KUKA KRL program: EPS_2_251315_MH05A_A_20251118013654.src

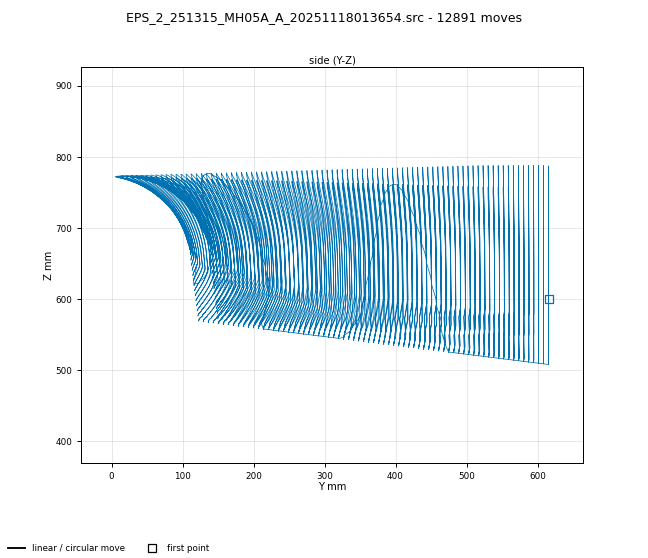
[picture p0: tool path of EPS_2_251315_MH05A_A_20251118013654.src, 12891 of 12893 moves have a stored position in this frame; points joined in program order, loops and branches not executed]
&ACCESS RVP
&REL 4
&COMMENT QRS 19112012
&PARAM EDITMASK = *
DEF PART()
EXT BAS (BAS_COMMAND :IN,REAL :IN )
INT I
BAS (#INITMOV,0 )

;KUKA QRS Post kuka4.cps  Date:22-06-2017 !

File_ID=2909

QRS_PRE_INIT()

;Init var - Until changes are made in qrs_pre_init
Outlet_Square_prg=0
Inlet_1_Square_prg=0
Inlet_2_Square_prg=0
Inlet_3_Square_prg=0
Inlet_4_Square_prg=0
Inlet_5_Square_prg=0

Outlet_1={X 0.000, Y 519.160, Z 687.500, B 0.000, E1 0.000 }
Inlet_1={X 0.000, Y 521.300, Z 657.500, B 0.000, E1 184.000 }
Outlet_1_type=201
Inlet_1_type=201
;QRS#1=Sidecore dimensions
;QRS#2=200-8" PVC SDR 35
;QRS#3=200-8" PVC SDR 35
;QRS#4=
;QRS#5=
;QRS#6=
;QRS#7=
;QRS#8=
;QRS#9=12-08 PSX
;QRS#10=12-08 PSX
;QRS#11=
;QRS#12=
;QRS#13=
;QRS#14=
;QRS#15=
;QRS#16=1220x127x1067 3,5'
;QRS#17=EPS Height
;QRS#18=788
;QRS#19=*
;QRS#20= UPDATED VERSION 22-06-2017
;QRS#21=*
Outlet_Square=0100
Inlet_1_Square=0100
Inlet_2_Square=0
Inlet_3_Square=0
Inlet_4_Square=0
Inlet_5_Square=0
Mill_Square=1
Outlet_Square_Prg=204
Inlet_1_Square_prg=204

QRS_INIT()

$ADVANCE=5

; T1
PTP {E1 173.595,E2 173.595}
PTP {X 0,Y 615.505,A -85,B 0,C 180,E1 173.595,E2 173.595,E3 0,E4 0,E5 0,E6 0}
QRS_SPEED_INIT()
LIN {X 0,Y 615.505,Z 600,A -85,B 0,C 180,E1 173.595,E2 173.595,E3 0,E4 0,E5 0,E6 0} C_VEL
LIN {X 0,Y 615.505,Z 517.862,A -85,B 0,C 180,E1 173.595,E2 173.595} C_VEL
LIN {X 0,Y 615.505,Z 509.682,A -85,B 0,C 180,E1 173.595,E2 173.595} C_VEL
LIN {X 0,Y 615.489,Z 507.682,A -85,B 0,C 180,E1 173.409,E2 173.409} C_VEL
LIN {X 0,Y 615.481,Z 507.696,A -85,B 0,C 180,E1 170.801,E2 170.801} C_VEL
LIN {X 0,Y 615.479,Z 507.691,A -85,B 0,C 180,E1 168.139,E2 168.139} C_VEL
LIN {X 0,Y 615.488,Z 507.682,A -85,B 0,C 180,E1 165.451,E2 165.451} C_VEL
LIN {X 0,Y 615.478,Z 507.699,A -85,B 0,C 180,E1 162.729,E2 162.729} C_VEL
LIN {X 0,Y 615.477,Z 507.687,A -85,B 0,C 180,E1 159.967,E2 159.967} C_VEL
LIN {X 0,Y 615.481,Z 507.683,A -85,B 0,C 180,E1 157.652,E2 157.652} C_VEL
LIN {X 0,Y 615.479,Z 507.691,A -85,B 0,C 180,E1 155.008,E2 155.008} C_VEL
LIN {X 0,Y 615.482,Z 507.688,A -85,B 0,C 180,E1 152.084,E2 152.084} C_VEL
LIN {X 0,Y 615.476,Z 507.686,A -85,B 0,C 180,E1 149.839,E2 149.839} C_VEL
LIN {X 0,Y 615.484,Z 507.683,A -85,B 0,C 180,E1 147.542,E2 147.542} C_VEL
LIN {X 0,Y 615.49,Z 507.685,A -85,B 0,C 180,E1 145.185,E2 145.185} C_VEL
LIN {X 0,Y 615.483,Z 507.698,A -85,B 0,C 180,E1 142.757,E2 142.757} C_VEL
LIN {X 0,Y 615.478,Z 507.686,A -85,B 0,C 180,E1 139.91,E2 139.91} C_VEL
LIN {X 0,Y 615.478,Z 507.684,A -85,B 0,C 180,E1 137.646,E2 137.646} C_VEL
LIN {X 0,Y 615.481,Z 507.693,A -85,B 0,C 180,E1 134.93,E2 134.93} C_VEL
LIN {X 0,Y 615.488,Z 507.687,A -85,B 0,C 180,E1 132.08,E2 132.08} C_VEL
LIN {X 0,Y 615.477,Z 507.685,A -85,B 0,C 180,E1 129.75,E2 129.75} C_VEL
LIN {X 0,Y 615.489,Z 507.691,A -85,B 0,C 180,E1 126.936,E2 126.936} C_VEL
LIN {X 0,Y 615.487,Z 507.686,A -85,B 0,C 180,E1 124.021,E2 124.021} C_VEL
LIN {X 0,Y 615.477,Z 507.684,A -85,B 0,C 180,E1 121.685,E2 121.685} C_VEL
LIN {X 0,Y 615.478,Z 507.685,A -85,B 0,C 180,E1 119.406,E2 119.406} C_VEL
LIN {X 0,Y 615.492,Z 507.688,A -85,B 0,C 180,E1 117.045,E2 117.045} C_VEL
LIN {X 0,Y 615.495,Z 507.689,A -85,B 0,C 180,E1 114.271,E2 114.271} C_VEL
LIN {X 0,Y 615.48,Z 507.684,A -85,B 0,C 180,E1 111.432,E2 111.432} C_VEL
LIN {X 0,Y 615.494,Z 507.701,A -85,B 0,C 180,E1 108.605,E2 108.605} C_VEL
LIN {X 0,Y 615.486,Z 507.684,A -85,B 0,C 180,E1 105.905,E2 105.905} C_VEL
LIN {X 0,Y 615.492,Z 507.887,A -85,B 0,C 180,E1 105.183,E2 105.183} C_VEL
LIN {X 0,Y 615.493,Z 525.05,A -85,B 0,C 180,E1 102.362,E2 102.362} C_VEL
LIN {X 0,Y 615.477,Z 542.524,A -85,B 0,C 180,E1 99.53,E2 99.53} C_VEL
LIN {X 0,Y 615.491,Z 546.889,A -85,B 0,C 180,E1 98.826,E2 98.826} C_VEL
LIN {X 0,Y 615.477,Z 653.781,A -85,B 0,C 180,E1 97.545,E2 97.545} C_VEL
LIN {X 0,Y 615.484,Z 666.943,A -85,B 0,C 180,E1 97.257,E2 97.257} C_VEL
LIN {X 0,Y 615.485,Z 679.264,A -85,B 0,C 180,E1 96.855,E2 96.855} C_VEL
LIN {X 0,Y 615.49,Z 691.591,A -85,B 0,C 180,E1 96.31,E2 96.31} C_VEL
LIN {X 0,Y 615.487,Z 702.986,A -85,B 0,C 180,E1 95.652,E2 95.652} C_VEL
LIN {X 0,Y 615.498,Z 713.247,A -85,B 0,C 180,E1 94.913,E2 94.913} C_VEL
LIN {X 0,Y 615.499,Z 722.526,A -85,B 0,C 180,E1 94.092,E2 94.092} C_VEL
LIN {X 0,Y 615.497,Z 731.469,A -85,B 0,C 180,E1 93.109,E2 93.109} C_VEL
LIN {X 0,Y 615.497,Z 738.692,A -85,B 0,C 180,E1 92.127,E2 92.127} C_VEL
LIN {X 0,Y 615.495,Z 745.319,A -85,B 0,C 180,E1 90.981,E2 90.981} C_VEL
LIN {X 0,Y 615.496,Z 749.706,A -85,B 0,C 180,E1 90,E2 90} C_VEL
LIN {X 0,Y 615.496,Z 752.021,A -85,B 0,C 180,E1 89.346,E2 89.346} C_VEL
LIN {X 0,Y 615.495,Z 753.917,A -85,B 0,C 180,E1 88.691,E2 88.691} C_VEL
LIN {X 0,Y 615.5,Z 755.401,A -85,B 0,C 180,E1 88.037,E2 88.037} C_VEL
LIN {X 0,Y 615.495,Z 757.09,A -85,B 0,C 180,E1 86.727,E2 86.727} C_VEL
LIN {X 0,Y 615.496,Z 757.254,A -85,B 0,C 180,E1 85.416,E2 85.416} C_VEL
LIN {X 0,Y 615.497,Z 755.79,A -85,B 0,C 180,E1 84.102,E2 84.102} C_VEL
LIN {X 0,Y 615.495,Z 754.424,A -85,B 0,C 180,E1 83.419,E2 83.419} C_VEL
LIN {X 0,Y 615.496,Z 751.671,A -85,B 0,C 180,E1 82.455,E2 82.455} C_VEL
LIN {X 0,Y 615.496,Z 747.841,A -85,B 0,C 180,E1 81.464,E2 81.464} C_VEL
LIN {X 0,Y 615.496,Z 742.869,A -85,B 0,C 180,E1 80.47,E2 80.47} C_VEL
LIN {X 0,Y 615.496,Z 736.598,A -85,B 0,C 180,E1 79.473,E2 79.473} C_VEL
LIN {X 0,Y 615.496,Z 728.708,A -85,B 0,C 180,E1 78.474,E2 78.474} C_VEL
LIN {X 0,Y 615.498,Z 720.622,A -85,B 0,C 180,E1 77.638,E2 77.638} C_VEL
LIN {X 0,Y 615.499,Z 710.724,A -85,B 0,C 180,E1 76.799,E2 76.799} C_VEL
LIN {X 0,Y 615.491,Z 699.961,A -85,B 0,C 180,E1 76.068,E2 76.068} C_VEL
LIN {X 0,Y 615.49,Z 688.509,A -85,B 0,C 180,E1 75.451,E2 75.451} C_VEL
LIN {X 0,Y 615.499,Z 676.28,A -85,B 0,C 180,E1 74.944,E2 74.944} C_VEL
LIN {X 0,Y 615.479,Z 663.455,A -85,B 0,C 180,E1 74.562,E2 74.562} C_VEL
LIN {X 0,Y 615.478,Z 649.799,A -85,B 0,C 180,E1 74.307,E2 74.307} C_VEL
LIN {X 0,Y 615.49,Z 546.948,A -85,B 0,C 180,E1 73.094,E2 73.094} C_VEL
LIN {X 0,Y 615.476,Z 529.77,A -85,B 0,C 180,E1 70.315,E2 70.315} C_VEL
LIN {X 0,Y 615.49,Z 513.503,A -85,B 0,C 180,E1 67.654,E2 67.654} C_VEL
LIN {X 0,Y 615.483,Z 507.686,A -85,B 0,C 180,E1 66.667,E2 66.667} C_VEL
LIN {X 0,Y 615.477,Z 507.684,A -85,B 0,C 180,E1 64.284,E2 64.284} C_VEL
LIN {X 0,Y 615.488,Z 507.694,A -85,B 0,C 180,E1 61.55,E2 61.55} C_VEL
LIN {X 0,Y 615.489,Z 507.689,A -85,B 0,C 180,E1 58.915,E2 58.915} C_VEL
LIN {X 0,Y 615.479,Z 507.684,A -85,B 0,C 180,E1 56.468,E2 56.468} C_VEL
LIN {X 0,Y 615.495,Z 507.692,A -85,B 0,C 180,E1 53.577,E2 53.577} C_VEL
LIN {X 0,Y 615.488,Z 507.69,A -85,B 0,C 180,E1 50.938,E2 50.938} C_VEL
LIN {X 0,Y 615.483,Z 507.684,A -85,B 0,C 180,E1 48.527,E2 48.527} C_VEL
LIN {X 0,Y 615.492,Z 507.686,A -85,B 0,C 180,E1 45.852,E2 45.852} C_VEL
LIN {X 0,Y 615.486,Z 507.693,A -85,B 0,C 180,E1 43.049,E2 43.049} C_VEL
LIN {X 0,Y 615.483,Z 507.684,A -85,B 0,C 180,E1 40.607,E2 40.607} C_VEL
LIN {X 0,Y 615.478,Z 507.686,A -85,B 0,C 180,E1 38.013,E2 38.013} C_VEL
LIN {X 0,Y 615.498,Z 507.691,A -85,B 0,C 180,E1 35.615,E2 35.615} C_VEL
LIN {X 0,Y 615.491,Z 507.698,A -85,B 0,C 180,E1 33.236,E2 33.236} C_VEL
LIN {X 0,Y 615.485,Z 507.69,A -85,B 0,C 180,E1 30.92,E2 30.92} C_VEL
LIN {X 0,Y 615.483,Z 507.683,A -85,B 0,C 180,E1 28.452,E2 28.452} C_VEL
LIN {X 0,Y 615.493,Z 507.693,A -85,B 0,C 180,E1 25.573,E2 25.573} C_VEL
LIN {X 0,Y 615.482,Z 507.688,A -85,B 0,C 180,E1 22.845,E2 22.845} C_VEL
LIN {X 0,Y 615.486,Z 507.683,A -85,B 0,C 180,E1 20.56,E2 20.56} C_VEL
LIN {X 0,Y 615.478,Z 507.687,A -85,B 0,C 180,E1 17.957,E2 17.957} C_VEL
LIN {X 0,Y 615.483,Z 507.699,A -85,B 0,C 180,E1 15.226,E2 15.226} C_VEL
LIN {X 0,Y 615.49,Z 507.682,A -85,B 0,C 180,E1 12.53,E2 12.53} C_VEL
LIN {X 0,Y 615.479,Z 507.689,A -85,B 0,C 180,E1 9.862,E2 9.862} C_VEL
LIN {X 0,Y 615.486,Z 507.697,A -85,B 0,C 180,E1 7.216,E2 7.216} C_VEL
LIN {X 0,Y 615.495,Z 507.681,A -85,B 0,C 180,E1 4.585,E2 4.585} C_VEL
LIN {X 0,Y 615.477,Z 507.688,A -85,B 0,C 180,E1 1.963,E2 1.963} C_VEL
LIN {X 0,Y 615.485,Z 507.702,A -85,B 0,C 180,E1 -0.654,E2 -0.654} C_VEL
LIN {X 0,Y 615.484,Z 507.685,A -85,B 0,C 180,E1 -3.273,E2 -3.273} C_VEL
LIN {X 0,Y 615.478,Z 507.686,A -85,B 0,C 180,E1 -5.899,E2 -5.899} C_VEL
LIN {X 0,Y 615.492,Z 507.699,A -85,B 0,C 180,E1 -8.537,E2 -8.537} C_VEL
LIN {X 0,Y 615.478,Z 507.687,A -85,B 0,C 180,E1 -11.193,E2 -11.193} C_VEL
LIN {X 0,Y 615.474,Z 507.687,A -85,B 0,C 180,E1 -13.933,E2 -13.933} C_VEL
LIN {X 0,Y 615.489,Z 507.702,A -85,B 0,C 180,E1 -16.587,E2 -16.587} C_VEL
LIN {X 0,Y 615.48,Z 507.685,A -85,B 0,C 180,E1 -19.338,E2 -19.338} C_VEL
LIN {X 0,Y 615.477,Z 507.691,A -85,B 0,C 180,E1 -22.137,E2 -22.137} C_VEL
LIN {X 0,Y 615.479,Z 507.691,A -85,B 0,C 180,E1 -24.992,E2 -24.992} C_VEL
LIN {X 0,Y 615.482,Z 507.686,A -85,B 0,C 180,E1 -27.915,E2 -27.915} C_VEL
LIN {X 0,Y 615.476,Z 507.692,A -85,B 0,C 180,E1 -30.161,E2 -30.161} C_VEL
LIN {X 0,Y 615.487,Z 507.699,A -85,B 0,C 180,E1 -32.458,E2 -32.458} C_VEL
LIN {X 0,Y 615.49,Z 507.693,A -85,B 0,C 180,E1 -34.815,E2 -34.815} C_VEL
LIN {X 0,Y 615.475,Z 507.687,A -85,B 0,C 180,E1 -37.243,E2 -37.243} C_VEL
LIN {X 0,Y 615.482,Z 507.689,A -85,B 0,C 180,E1 -40.09,E2 -40.09} C_VEL
LIN {X 0,Y 615.478,Z 507.697,A -85,B 0,C 180,E1 -42.354,E2 -42.354} C_VEL
LIN {X 0,Y 615.48,Z 507.689,A -85,B 0,C 180,E1 -45.069,E2 -45.069} C_VEL
LIN {X 0,Y 615.488,Z 507.685,A -85,B 0,C 180,E1 -47.92,E2 -47.92} C_VEL
LIN {X 0,Y 615.48,Z 507.694,A -85,B 0,C 180,E1 -50.25,E2 -50.25} C_VEL
LIN {X 0,Y 615.482,Z 507.688,A -85,B 0,C 180,E1 -53.064,E2 -53.064} C_VEL
LIN {X 0,Y 615.487,Z 507.686,A -85,B 0,C 180,E1 -55.979,E2 -55.979} C_VEL
LIN {X 0,Y 615.489,Z 507.69,A -85,B 0,C 180,E1 -58.914,E2 -58.914} C_VEL
LIN {X 0,Y 615.481,Z 507.683,A -85,B 0,C 180,E1 -61.551,E2 -61.551} C_VEL
LIN {X 0,Y 615.477,Z 507.696,A -85,B 0,C 180,E1 -64.284,E2 -64.284} C_VEL
LIN {X 0,Y 615.486,Z 507.7,A -85,B 0,C 180,E1 -66.444,E2 -66.444} C_VEL
LIN {X 0,Y 615.491,Z 507.764,A -85,B 0,C 180,E1 -67.838,E2 -67.838} C_VEL
LIN {X 0,Y 615.483,Z 528.08,A -85,B 0,C 180,E1 -70.662,E2 -70.662} C_VEL
LIN {X 0,Y 615.477,Z 548.189,A -85,B 0,C 180,E1 -73.414,E2 -73.414} C_VEL
LIN {X 0,Y 615.487,Z 568.274,A -85,B 0,C 180,E1 -76.126,E2 -76.126} C_VEL
LIN {X 0,Y 615.486,Z 575.644,A -85,B 0,C 180,E1 -77.114,E2 -77.114} C_VEL
LIN {X 0,Y 615.477,Z 683.848,A -85,B 0,C 180,E1 -78.411,E2 -78.411} C_VEL
LIN {X 0,Y 615.482,Z 696.355,A -85,B 0,C 180,E1 -78.682,E2 -78.682} C_VEL
LIN {X 0,Y 615.497,Z 709.489,A -85,B 0,C 180,E1 -79.108,E2 -79.108} C_VEL
LIN {X 0,Y 615.48,Z 721.483,A -85,B 0,C 180,E1 -79.64,E2 -79.64} C_VEL
LIN {X 0,Y 615.481,Z 733,A -85,B 0,C 180,E1 -80.304,E2 -80.304} C_VEL
LIN {X 0,Y 615.499,Z 743.344,A -85,B 0,C 180,E1 -81.05,E2 -81.05} C_VEL
LIN {X 0,Y 615.497,Z 751.814,A -85,B 0,C 180,E1 -81.794,E2 -81.794} C_VEL
LIN {X 0,Y 615.498,Z 759.608,A -85,B 0,C 180,E1 -82.62,E2 -82.62} C_VEL
LIN {X 0,Y 615.496,Z 767.204,A -85,B 0,C 180,E1 -83.608,E2 -83.608} C_VEL
LIN {X 0,Y 615.498,Z 774.205,A -85,B 0,C 180,E1 -84.759,E2 -84.759} C_VEL
LIN {X 0,Y 615.493,Z 778.852,A -85,B 0,C 180,E1 -85.744,E2 -85.744} C_VEL
LIN {X 0,Y 615.495,Z 782.399,A -85,B 0,C 180,E1 -86.727,E2 -86.727} C_VEL
LIN {X 0,Y 615.497,Z 784.233,A -85,B 0,C 180,E1 -87.382,E2 -87.382} C_VEL
LIN {X 0,Y 615.496,Z 785.608,A -85,B 0,C 180,E1 -88.037,E2 -88.037} C_VEL
LIN {X 0,Y 615.496,Z 787.174,A -85,B 0,C 180,E1 -89.346,E2 -89.346} C_VEL
LIN {X 0,Y 615.494,Z 787.389,A -85,B 0,C 180,E1 -90,E2 -90} C_VEL
LIN {X 0,Y 615.496,Z 786.58,A -85,B 0,C 180,E1 -91.309,E2 -91.309} C_VEL
LIN {X 0,Y 615.496,Z 785.608,A -85,B 0,C 180,E1 -91.963,E2 -91.963} C_VEL
LIN {X 0,Y 615.497,Z 784.233,A -85,B 0,C 180,E1 -92.618,E2 -92.618} C_VEL
LIN {X 0,Y 615.496,Z 781.35,A -85,B 0,C 180,E1 -93.601,E2 -93.601} C_VEL
LIN {X 0,Y 615.498,Z 777.442,A -85,B 0,C 180,E1 -94.584,E2 -94.584} C_VEL
LIN {X 0,Y 615.499,Z 772.406,A -85,B 0,C 180,E1 -95.57,E2 -95.57} C_VEL
LIN {X 0,Y 615.497,Z 765.869,A -85,B 0,C 180,E1 -96.583,E2 -96.583} C_VEL
LIN {X 0,Y 615.497,Z 758.135,A -85,B 0,C 180,E1 -97.545,E2 -97.545} C_VEL
LIN {X 0,Y 615.498,Z 750.047,A -85,B 0,C 180,E1 -98.371,E2 -98.371} C_VEL
LIN {X 0,Y 615.499,Z 740.17,A -85,B 0,C 180,E1 -99.198,E2 -99.198} C_VEL
LIN {X 0,Y 615.483,Z 728.986,A -85,B 0,C 180,E1 -99.945,E2 -99.945} C_VEL
LIN {X 0,Y 615.481,Z 718.029,A -85,B 0,C 180,E1 -100.527,E2 -100.527} C_VEL
LIN {X 0,Y 615.499,Z 705.423,A -85,B 0,C 180,E1 -101.042,E2 -101.042} C_VEL
LIN {X 0,Y 615.479,Z 693.079,A -85,B 0,C 180,E1 -101.401,E2 -101.401} C_VEL
LIN {X 0,Y 615.477,Z 679.489,A -85,B 0,C 180,E1 -101.652,E2 -101.652} C_VEL
LIN {X 0,Y 615.486,Z 575.644,A -85,B 0,C 180,E1 -102.886,E2 -102.886} C_VEL
LIN {X 0,Y 615.479,Z 554.469,A -85,B 0,C 180,E1 -105.735,E2 -105.735} C_VEL
LIN {X 0,Y 615.479,Z 534.609,A -85,B 0,C 180,E1 -108.44,E2 -108.44} C_VEL
LIN {X 0,Y 615.497,Z 514.243,A -85,B 0,C 180,E1 -111.255,E2 -111.255} C_VEL
LIN {X 0,Y 615.489,Z 507.683,A -85,B 0,C 180,E1 -112.188,E2 -112.188} C_VEL
LIN {X 0,Y 615.488,Z 507.687,A -85,B 0,C 180,E1 -114.991,E2 -114.991} C_VEL
LIN {X 0,Y 615.483,Z 507.69,A -85,B 0,C 180,E1 -117.915,E2 -117.915} C_VEL
LIN {X 0,Y 615.499,Z 507.681,A -85,B 0,C 180,E1 -120.159,E2 -120.159} C_VEL
LIN {X 0,Y 615.481,Z 507.683,A -85,B 0,C 180,E1 -122.457,E2 -122.457} C_VEL
LIN {X 0,Y 615.478,Z 507.686,A -85,B 0,C 180,E1 -124.815,E2 -124.815} C_VEL
LIN {X 0,Y 615.496,Z 507.693,A -85,B 0,C 180,E1 -127.241,E2 -127.241} C_VEL
LIN {X 0,Y 615.49,Z 507.684,A -85,B 0,C 180,E1 -130.089,E2 -130.089} C_VEL
LIN {X 0,Y 615.49,Z 507.681,A -85,B 0,C 180,E1 -132.351,E2 -132.351} C_VEL
LIN {X 0,Y 615.481,Z 507.691,A -85,B 0,C 180,E1 -135.068,E2 -135.068} C_VEL
LIN {X 0,Y 615.477,Z 507.69,A -85,B 0,C 180,E1 -137.919,E2 -137.919} C_VEL
LIN {X 0,Y 615.498,Z 507.68,A -85,B 0,C 180,E1 -140.251,E2 -140.251} C_VEL
LIN {X 0,Y 615.48,Z 507.691,A -85,B 0,C 180,E1 -143.063,E2 -143.063} C_VEL
LIN {X 0,Y 615.494,Z 507.695,A -85,B 0,C 180,E1 -145.297,E2 -145.297} C_VEL
LIN {X 0,Y 615.485,Z 507.683,A -85,B 0,C 180,E1 -148.314,E2 -148.314} C_VEL
LIN {X 0,Y 615.482,Z 507.683,A -85,B 0,C 180,E1 -150.593,E2 -150.593} C_VEL
LIN {X 0,Y 615.478,Z 507.689,A -85,B 0,C 180,E1 -152.954,E2 -152.954} C_VEL
LIN {X 0,Y 615.478,Z 507.695,A -85,B 0,C 180,E1 -155.728,E2 -155.728} C_VEL
LIN {X 0,Y 615.486,Z 507.682,A -85,B 0,C 180,E1 -158.568,E2 -158.568} C_VEL
LIN {X 0,Y 615.495,Z 507.699,A -85,B 0,C 180,E1 -161.389,E2 -161.389} C_VEL
LIN {X 0,Y 615.48,Z 507.686,A -85,B 0,C 180,E1 -164.095,E2 -164.095} C_VEL
LIN {X 0,Y 615.478,Z 507.687,A -85,B 0,C 180,E1 -166.799,E2 -166.799} C_VEL
LIN {X 0,Y 615.488,Z 507.701,A -85,B 0,C 180,E1 -169.473,E2 -169.473} C_VEL
LIN {X 0,Y 615.479,Z 507.686,A -85,B 0,C 180,E1 -172.124,E2 -172.124} C_VEL
LIN {X 0,Y 615.481,Z 507.685,A -85,B 0,C 180,E1 -174.759,E2 -174.759} C_VEL
LIN {X 0,Y 615.495,Z 507.699,A -85,B 0,C 180,E1 -177.382,E2 -177.382} C_VEL
LIN {X 0,Y 615.477,Z 507.688,A -85,B 0,C 180,E1 -180,E2 -180} C_VEL
LIN {X 0,Y 615.492,Z 507.682,A -85,B 0,C 180,E1 -182.618,E2 -182.618} C_VEL
LIN {X 0,Y 615.481,Z 507.697,A -85,B 0,C 180,E1 -185.241,E2 -185.241} C_VEL
LIN {X 0,Y 615.489,Z 507.682,A -85,B 0,C 180,E1 -186.591,E2 -186.591} C_VEL
LIN {X 0,Y 614.809,Z 507.843,A -85,B 0,C 180,E1 -187.137,E2 -187.137} C_VEL
LIN {X 0,Y 611.97,Z 508.251,A -85,B 0,C 180,E1 -188.023,E2 -188.023} C_VEL
LIN {X 0,Y 609.577,Z 508.566,A -85,B 0,C 180,E1 -188.735,E2 -188.735} C_VEL
LIN {X 0,Y 608.542,Z 508.685,A -85,B 0,C 180,E1 -189.285,E2 -189.285} C_VEL
LIN {X 0,Y 608.452,Z 508.693,A -85,B 0,C 180,E1 -189.471,E2 -189.471} C_VEL
LIN {X 0,Y 608.456,Z 508.689,A -85,B 0,C 180,E1 -192,E2 -192} C_VEL
LIN {X 0,Y 608.474,Z 508.685,A -85,B 0,C 180,E1 -194.721,E2 -194.721} C_VEL
LIN {X 0,Y 608.445,Z 508.698,A -85,B 0,C 180,E1 -197.477,E2 -197.477} C_VEL
LIN {X 0,Y 608.458,Z 508.687,A -85,B 0,C 180,E1 -200.275,E2 -200.275} C_VEL
LIN {X 0,Y 608.449,Z 508.687,A -85,B 0,C 180,E1 -202.477,E2 -202.477} C_VEL
LIN {X 0,Y 608.453,Z 508.696,A -85,B 0,C 180,E1 -205.301,E2 -205.301} C_VEL
LIN {X 0,Y 608.446,Z 508.697,A -85,B 0,C 180,E1 -207.518,E2 -207.518} C_VEL
LIN {X 0,Y 608.465,Z 508.688,A -85,B 0,C 180,E1 -209.973,E2 -209.973} C_VEL
LIN {X 0,Y 608.458,Z 508.686,A -85,B 0,C 180,E1 -212.524,E2 -212.524} C_VEL
LIN {X 0,Y 608.453,Z 508.696,A -85,B 0,C 180,E1 -215.277,E2 -215.277} C_VEL
LIN {X 0,Y 608.464,Z 508.691,A -85,B 0,C 180,E1 -217.747,E2 -217.747} C_VEL
LIN {X 0,Y 608.446,Z 508.688,A -85,B 0,C 180,E1 -220.33,E2 -220.33} C_VEL
LIN {X 0,Y 608.467,Z 508.695,A -85,B 0,C 180,E1 -223.31,E2 -223.31} C_VEL
LIN {X 0,Y 608.469,Z 508.686,A -85,B 0,C 180,E1 -226.132,E2 -226.132} C_VEL
LIN {X 0,Y 608.452,Z 508.689,A -85,B 0,C 180,E1 -228.824,E2 -228.824} C_VEL
LIN {X 0,Y 608.468,Z 508.696,A -85,B 0,C 180,E1 -231.413,E2 -231.413} C_VEL
LIN {X 0,Y 608.458,Z 508.689,A -85,B 0,C 180,E1 -233.954,E2 -233.954} C_VEL
LIN {X 0,Y 608.449,Z 508.688,A -85,B 0,C 180,E1 -236.329,E2 -236.329} C_VEL
LIN {X 0,Y 608.461,Z 508.687,A -85,B 0,C 180,E1 -238.731,E2 -238.731} C_VEL
LIN {X 0,Y 608.475,Z 508.695,A -85,B 0,C 180,E1 -241.381,E2 -241.381} C_VEL
LIN {X 0,Y 608.443,Z 508.69,A -85,B 0,C 180,E1 -243.965,E2 -243.965} C_VEL
LIN {X 0,Y 608.467,Z 508.686,A -85,B 0,C 180,E1 -246.156,E2 -246.156} C_VEL
LIN {X 0,Y 608.469,Z 508.685,A -85,B 0,C 180,E1 -248.309,E2 -248.309} C_VEL
LIN {X 0,Y 608.477,Z 508.693,A -85,B 0,C 180,E1 -251.284,E2 -251.284} C_VEL
LIN {X 0,Y 608.463,Z 508.689,A -85,B 0,C 180,E1 -253.907,E2 -253.907} C_VEL
LIN {X 0,Y 608.483,Z 508.758,A -85,B 0,C 180,E1 -254.723,E2 -254.723} C_VEL
LIN {X 0,Y 608.493,Z 525.455,A -85,B 0,C 180,E1 -257.493,E2 -257.493} C_VEL
LIN {X 0,Y 608.473,Z 541.956,A -85,B 0,C 180,E1 -260.191,E2 -260.191} C_VEL
LIN {X 0,Y 608.475,Z 547.189,A -85,B 0,C 180,E1 -261.04,E2 -261.04} C_VEL
LIN {X 0,Y 608.523,Z 654.213,A -85,B 0,C 180,E1 -262.326,E2 -262.326} C_VEL
LIN {X 0,Y 608.519,Z 667.268,A -85,B 0,C 180,E1 -262.618,E2 -262.618} C_VEL
LIN {X 0,Y 608.509,Z 680.713,A -85,B 0,C 180,E1 -263.068,E2 -263.068} C_VEL
LIN {X 0,Y 608.502,Z 692.957,A -85,B 0,C 180,E1 -263.635,E2 -263.635} C_VEL
LIN {X 0,Y 608.485,Z 703.909,A -85,B 0,C 180,E1 -264.283,E2 -264.283} C_VEL
LIN {X 0,Y 608.476,Z 714.098,A -85,B 0,C 180,E1 -265.031,E2 -265.031} C_VEL
LIN {X 0,Y 608.473,Z 723.296,A -85,B 0,C 180,E1 -265.86,E2 -265.86} C_VEL
LIN {X 0,Y 608.459,Z 732.223,A -85,B 0,C 180,E1 -266.855,E2 -266.855} C_VEL
LIN {X 0,Y 608.454,Z 739.435,A -85,B 0,C 180,E1 -267.849,E2 -267.849} C_VEL
LIN {X 0,Y 608.449,Z 744.316,A -85,B 0,C 180,E1 -268.676,E2 -268.676} C_VEL
LIN {X 0,Y 608.442,Z 749.071,A -85,B 0,C 180,E1 -269.669,E2 -269.669} C_VEL
LIN {X 0,Y 608.439,Z 752.725,A -85,B 0,C 180,E1 -270.662,E2 -270.662} C_VEL
LIN {X 0,Y 608.447,Z 754.616,A -85,B 0,C 180,E1 -271.324,E2 -271.324} C_VEL
LIN {X 0,Y 608.445,Z 756.078,A -85,B 0,C 180,E1 -271.986,E2 -271.986} C_VEL
LIN {X 0,Y 608.421,Z 757.733,A -85,B 0,C 180,E1 -273.311,E2 -273.311} C_VEL
LIN {X 0,Y 608.433,Z 757.989,A -85,B 0,C 180,E1 -273.974,E2 -273.974} C_VEL
LIN {X 0,Y 608.429,Z 757.832,A -85,B 0,C 180,E1 -274.638,E2 -274.638} C_VEL
LIN {X 0,Y 608.434,Z 756.307,A -85,B 0,C 180,E1 -275.967,E2 -275.967} C_VEL
LIN {X 0,Y 608.448,Z 754.954,A -85,B 0,C 180,E1 -276.633,E2 -276.633} C_VEL
LIN {X 0,Y 608.427,Z 752.071,A -85,B 0,C 180,E1 -277.633,E2 -277.633} C_VEL
LIN {X 0,Y 608.43,Z 748.15,A -85,B 0,C 180,E1 -278.636,E2 -278.636} C_VEL
LIN {X 0,Y 608.435,Z 743.074,A -85,B 0,C 180,E1 -279.642,E2 -279.642} C_VEL
LIN {X 0,Y 608.443,Z 736.674,A -85,B 0,C 180,E1 -280.65,E2 -280.65} C_VEL
LIN {X 0,Y 608.474,Z 728.627,A -85,B 0,C 180,E1 -281.661,E2 -281.661} C_VEL
LIN {X 0,Y 608.468,Z 720.403,A -85,B 0,C 180,E1 -282.507,E2 -282.507} C_VEL
LIN {X 0,Y 608.481,Z 710.336,A -85,B 0,C 180,E1 -283.356,E2 -283.356} C_VEL
LIN {X 0,Y 608.489,Z 698.896,A -85,B 0,C 180,E1 -284.122,E2 -284.122} C_VEL
LIN {X 0,Y 608.518,Z 687.649,A -85,B 0,C 180,E1 -284.719,E2 -284.719} C_VEL
LIN {X 0,Y 608.545,Z 675.035,A -85,B 0,C 180,E1 -285.232,E2 -285.232} C_VEL
LIN {X 0,Y 608.545,Z 662.387,A -85,B 0,C 180,E1 -285.597,E2 -285.597} C_VEL
LIN {X 0,Y 608.547,Z 649.513,A -85,B 0,C 180,E1 -285.833,E2 -285.833} C_VEL
LIN {X 0,Y 608.467,Z 547.168,A -85,B 0,C 180,E1 -287.053,E2 -287.053} C_VEL
LIN {X 0,Y 608.488,Z 529.572,A -85,B 0,C 180,E1 -289.92,E2 -289.92} C_VEL
LIN {X 0,Y 608.512,Z 512.592,A -85,B 0,C 180,E1 -292.726,E2 -292.726} C_VEL
LIN {X 0,Y 608.464,Z 508.688,A -85,B 0,C 180,E1 -293.393,E2 -293.393} C_VEL
LIN {X 0,Y 608.443,Z 508.69,A -85,B 0,C 180,E1 -296.035,E2 -296.035} C_VEL
LIN {X 0,Y 608.475,Z 508.694,A -85,B 0,C 180,E1 -298.619,E2 -298.619} C_VEL
LIN {X 0,Y 608.46,Z 508.688,A -85,B 0,C 180,E1 -301.316,E2 -301.316} C_VEL
LIN {X 0,Y 608.471,Z 508.685,A -85,B 0,C 180,E1 -303.734,E2 -303.734} C_VEL
LIN {X 0,Y 608.476,Z 508.686,A -85,B 0,C 180,E1 -306.089,E2 -306.089} C_VEL
LIN {X 0,Y 608.468,Z 508.694,A -85,B 0,C 180,E1 -308.587,E2 -308.587} C_VEL
LIN {X 0,Y 608.458,Z 508.688,A -85,B 0,C 180,E1 -311.341,E2 -311.341} C_VEL
LIN {X 0,Y 608.459,Z 508.69,A -85,B 0,C 180,E1 -314.264,E2 -314.264} C_VEL
LIN {X 0,Y 608.452,Z 508.692,A -85,B 0,C 180,E1 -317.04,E2 -317.04} C_VEL
LIN {X 0,Y 608.446,Z 508.688,A -85,B 0,C 180,E1 -319.696,E2 -319.696} C_VEL
LIN {X 0,Y 608.463,Z 508.69,A -85,B 0,C 180,E1 -322.253,E2 -322.253} C_VEL
LIN {X 0,Y 608.481,Z 508.687,A -85,B 0,C 180,E1 -325.088,E2 -325.088} C_VEL
LIN {X 0,Y 608.463,Z 508.686,A -85,B 0,C 180,E1 -327.905,E2 -327.905} C_VEL
LIN {X 0,Y 608.472,Z 508.688,A -85,B 0,C 180,E1 -330.22,E2 -330.22} C_VEL
LIN {X 0,Y 608.474,Z 508.693,A -85,B 0,C 180,E1 -332.791,E2 -332.791} C_VEL
LIN {X 0,Y 608.445,Z 508.688,A -85,B 0,C 180,E1 -335.428,E2 -335.428} C_VEL
LIN {X 0,Y 608.471,Z 508.69,A -85,B 0,C 180,E1 -338.308,E2 -338.308} C_VEL
LIN {X 0,Y 608.469,Z 508.686,A -85,B 0,C 180,E1 -341.28,E2 -341.28} C_VEL
LIN {X 0,Y 608.456,Z 508.687,A -85,B 0,C 180,E1 -343.906,E2 -343.906} C_VEL
LIN {X 0,Y 608.457,Z 508.698,A -85,B 0,C 180,E1 -346.643,E2 -346.643} C_VEL
LIN {X 0,Y 608.463,Z 508.687,A -85,B 0,C 180,E1 -349.35,E2 -349.35} C_VEL
LIN {X 0,Y 608.471,Z 508.687,A -85,B 0,C 180,E1 -352.033,E2 -352.033} C_VEL
LIN {X 0,Y 608.461,Z 508.696,A -85,B 0,C 180,E1 -354.698,E2 -354.698} C_VEL
LIN {X 0,Y 608.481,Z 508.684,A -85,B 0,C 180,E1 -357.352,E2 -357.352} C_VEL
LIN {X 0,Y 608.467,Z 508.687,A -85,B 0,C 180,E1 -360,E2 -360} C_VEL
LIN {X 0,Y 608.484,Z 508.694,A -85,B 0,C 180,E1 -362.648,E2 -362.648} C_VEL
LIN {X 0,Y 608.46,Z 508.687,A -85,B 0,C 180,E1 -365.302,E2 -365.302} C_VEL
LIN {X 0,Y 608.472,Z 508.686,A -85,B 0,C 180,E1 -367.967,E2 -367.967} C_VEL
LIN {X 0,Y 608.463,Z 508.696,A -85,B 0,C 180,E1 -370.65,E2 -370.65} C_VEL
LIN {X 0,Y 608.455,Z 508.687,A -85,B 0,C 180,E1 -373.357,E2 -373.357} C_VEL
LIN {X 0,Y 608.455,Z 508.69,A -85,B 0,C 180,E1 -376.094,E2 -376.094} C_VEL
LIN {X 0,Y 608.452,Z 508.693,A -85,B 0,C 180,E1 -378.87,E2 -378.87} C_VEL
LIN {X 0,Y 608.464,Z 508.686,A -85,B 0,C 180,E1 -381.692,E2 -381.692} C_VEL
LIN {X 0,Y 608.445,Z 508.699,A -85,B 0,C 180,E1 -384.571,E2 -384.571} C_VEL
LIN {X 0,Y 608.47,Z 508.686,A -85,B 0,C 180,E1 -387.208,E2 -387.208} C_VEL
LIN {X 0,Y 608.464,Z 508.687,A -85,B 0,C 180,E1 -389.973,E2 -389.973} C_VEL
LIN {X 0,Y 608.46,Z 508.697,A -85,B 0,C 180,E1 -392.524,E2 -392.524} C_VEL
LIN {X 0,Y 608.449,Z 508.688,A -85,B 0,C 180,E1 -395.277,E2 -395.277} C_VEL
LIN {X 0,Y 608.462,Z 508.686,A -85,B 0,C 180,E1 -397.747,E2 -397.747} C_VEL
LIN {X 0,Y 608.45,Z 508.694,A -85,B 0,C 180,E1 -400.33,E2 -400.33} C_VEL
LIN {X 0,Y 608.463,Z 508.686,A -85,B 0,C 180,E1 -403.31,E2 -403.31} C_VEL
LIN {X 0,Y 608.471,Z 508.689,A -85,B 0,C 180,E1 -406.132,E2 -406.132} C_VEL
LIN {X 0,Y 608.458,Z 508.692,A -85,B 0,C 180,E1 -408.825,E2 -408.825} C_VEL
LIN {X 0,Y 608.465,Z 508.686,A -85,B 0,C 180,E1 -411.413,E2 -411.413} C_VEL
LIN {X 0,Y 608.457,Z 508.688,A -85,B 0,C 180,E1 -413.953,E2 -413.953} C_VEL
LIN {X 0,Y 608.467,Z 508.693,A -85,B 0,C 180,E1 -416.33,E2 -416.33} C_VEL
LIN {X 0,Y 608.477,Z 508.691,A -85,B 0,C 180,E1 -418.728,E2 -418.728} C_VEL
LIN {X 0,Y 608.467,Z 508.686,A -85,B 0,C 180,E1 -421.382,E2 -421.382} C_VEL
LIN {X 0,Y 608.438,Z 508.691,A -85,B 0,C 180,E1 -423.965,E2 -423.965} C_VEL
LIN {X 0,Y 608.469,Z 508.69,A -85,B 0,C 180,E1 -426.156,E2 -426.156} C_VEL
LIN {X 0,Y 608.472,Z 508.737,A -85,B 0,C 180,E1 -427.707,E2 -427.707} C_VEL
LIN {X 0,Y 608.535,Z 524.321,A -85,B 0,C 180,E1 -429.905,E2 -429.905} C_VEL
LIN {X 0,Y 608.527,Z 544.47,A -85,B 0,C 180,E1 -432.699,E2 -432.699} C_VEL
LIN {X 0,Y 608.497,Z 565.878,A -85,B 0,C 180,E1 -435.622,E2 -435.622} C_VEL
LIN {X 0,Y 608.495,Z 576.169,A -85,B 0,C 180,E1 -436.984,E2 -436.984} C_VEL
LIN {X 0,Y 608.534,Z 683.962,A -85,B 0,C 180,E1 -438.277,E2 -438.277} C_VEL
LIN {X 0,Y 608.533,Z 697.226,A -85,B 0,C 180,E1 -438.572,E2 -438.572} C_VEL
LIN {X 0,Y 608.544,Z 710.334,A -85,B 0,C 180,E1 -439.009,E2 -439.009} C_VEL
LIN {X 0,Y 608.498,Z 721.64,A -85,B 0,C 180,E1 -439.519,E2 -439.519} C_VEL
LIN {X 0,Y 608.471,Z 733.201,A -85,B 0,C 180,E1 -440.191,E2 -440.191} C_VEL
LIN {X 0,Y 608.485,Z 743.596,A -85,B 0,C 180,E1 -440.946,E2 -440.946} C_VEL
LIN {X 0,Y 608.475,Z 752.114,A -85,B 0,C 180,E1 -441.699,E2 -441.699} C_VEL
LIN {X 0,Y 608.471,Z 759.962,A -85,B 0,C 180,E1 -442.534,E2 -442.534} C_VEL
LIN {X 0,Y 608.46,Z 767.287,A -85,B 0,C 180,E1 -443.485,E2 -443.485} C_VEL
LIN {X 0,Y 608.45,Z 772.867,A -85,B 0,C 180,E1 -444.366,E2 -444.366} C_VEL
LIN {X 0,Y 608.432,Z 777.951,A -85,B 0,C 180,E1 -445.362,E2 -445.362} C_VEL
LIN {X 0,Y 608.449,Z 781.896,A -85,B 0,C 180,E1 -446.358,E2 -446.358} C_VEL
LIN {X 0,Y 608.425,Z 784.809,A -85,B 0,C 180,E1 -447.352,E2 -447.352} C_VEL
LIN {X 0,Y 608.441,Z 786.201,A -85,B 0,C 180,E1 -448.014,E2 -448.014} C_VEL
LIN {X 0,Y 608.438,Z 787.783,A -85,B 0,C 180,E1 -449.338,E2 -449.338} C_VEL
LIN {X 0,Y 608.434,Z 788,A -85,B 0,C 180,E1 -450,E2 -450} C_VEL
LIN {X 0,Y 608.448,Z 787.184,A -85,B 0,C 180,E1 -451.324,E2 -451.324} C_VEL
LIN {X 0,Y 608.441,Z 786.201,A -85,B 0,C 180,E1 -451.986,E2 -451.986} C_VEL
LIN {X 0,Y 608.425,Z 784.809,A -85,B 0,C 180,E1 -452.648,E2 -452.648} C_VEL
LIN {X 0,Y 608.449,Z 781.896,A -85,B 0,C 180,E1 -453.642,E2 -453.642} C_VEL
LIN {X 0,Y 608.432,Z 777.951,A -85,B 0,C 180,E1 -454.638,E2 -454.638} C_VEL
LIN {X 0,Y 608.437,Z 771.877,A -85,B 0,C 180,E1 -455.801,E2 -455.801} C_VEL
LIN {X 0,Y 608.462,Z 765.236,A -85,B 0,C 180,E1 -456.799,E2 -456.799} C_VEL
LIN {X 0,Y 608.455,Z 756.991,A -85,B 0,C 180,E1 -457.8,E2 -457.8} C_VEL
LIN {X 0,Y 608.472,Z 748.539,A -85,B 0,C 180,E1 -458.636,E2 -458.636} C_VEL
LIN {X 0,Y 608.474,Z 738.094,A -85,B 0,C 180,E1 -459.473,E2 -459.473} C_VEL
LIN {X 0,Y 608.482,Z 727.76,A -85,B 0,C 180,E1 -460.145,E2 -460.145} C_VEL
LIN {X 0,Y 608.521,Z 716.245,A -85,B 0,C 180,E1 -460.741,E2 -460.741} C_VEL
LIN {X 0,Y 608.528,Z 704.882,A -85,B 0,C 180,E1 -461.192,E2 -461.192} C_VEL
LIN {X 0,Y 608.535,Z 692.279,A -85,B 0,C 180,E1 -461.554,E2 -461.554} C_VEL
LIN {X 0,Y 608.535,Z 679.622,A -85,B 0,C 180,E1 -461.787,E2 -461.787} C_VEL
LIN {X 0,Y 608.495,Z 576.169,A -85,B 0,C 180,E1 -463.016,E2 -463.016} C_VEL
LIN {X 0,Y 608.487,Z 557.063,A -85,B 0,C 180,E1 -465.577,E2 -465.577} C_VEL
LIN {X 0,Y 608.516,Z 536.995,A -85,B 0,C 180,E1 -468.332,E2 -468.332} C_VEL
LIN {X 0,Y 608.572,Z 516.765,A -85,B 0,C 180,E1 -471.154,E2 -471.154} C_VEL
LIN {X 0,Y 608.455,Z 508.689,A -85,B 0,C 180,E1 -472.316,E2 -472.316} C_VEL
LIN {X 0,Y 608.455,Z 508.687,A -85,B 0,C 180,E1 -474.57,E2 -474.57} C_VEL
LIN {X 0,Y 608.484,Z 508.689,A -85,B 0,C 180,E1 -477.208,E2 -477.208} C_VEL
LIN {X 0,Y 608.467,Z 508.688,A -85,B 0,C 180,E1 -479.971,E2 -479.971} C_VEL
LIN {X 0,Y 608.457,Z 508.686,A -85,B 0,C 180,E1 -482.521,E2 -482.521} C_VEL
LIN {X 0,Y 608.443,Z 508.69,A -85,B 0,C 180,E1 -484.904,E2 -484.904} C_VEL
LIN {X 0,Y 608.471,Z 508.691,A -85,B 0,C 180,E1 -487.745,E2 -487.745} C_VEL
LIN {X 0,Y 608.45,Z 508.688,A -85,B 0,C 180,E1 -490.329,E2 -490.329} C_VEL
LIN {X 0,Y 608.485,Z 508.691,A -85,B 0,C 180,E1 -493.31,E2 -493.31} C_VEL
LIN {X 0,Y 608.466,Z 508.687,A -85,B 0,C 180,E1 -496.13,E2 -496.13} C_VEL
LIN {X 0,Y 608.449,Z 508.689,A -85,B 0,C 180,E1 -498.823,E2 -498.823} C_VEL
LIN {X 0,Y 608.465,Z 508.696,A -85,B 0,C 180,E1 -501.412,E2 -501.412} C_VEL
LIN {X 0,Y 608.472,Z 508.688,A -85,B 0,C 180,E1 -503.949,E2 -503.949} C_VEL
LIN {X 0,Y 608.462,Z 508.686,A -85,B 0,C 180,E1 -506.329,E2 -506.329} C_VEL
LIN {X 0,Y 608.469,Z 508.686,A -85,B 0,C 180,E1 -508.727,E2 -508.727} C_VEL
LIN {X 0,Y 608.471,Z 508.695,A -85,B 0,C 180,E1 -511.378,E2 -511.378} C_VEL
LIN {X 0,Y 608.475,Z 508.685,A -85,B 0,C 180,E1 -514.276,E2 -514.276} C_VEL
LIN {X 0,Y 608.447,Z 508.69,A -85,B 0,C 180,E1 -516.876,E2 -516.876} C_VEL
LIN {X 0,Y 608.464,Z 508.694,A -85,B 0,C 180,E1 -519.319,E2 -519.319} C_VEL
LIN {X 0,Y 608.448,Z 508.692,A -85,B 0,C 180,E1 -521.828,E2 -521.828} C_VEL
LIN {X 0,Y 608.463,Z 508.686,A -85,B 0,C 180,E1 -524.594,E2 -524.594} C_VEL
LIN {X 0,Y 608.473,Z 508.693,A -85,B 0,C 180,E1 -527.323,E2 -527.323} C_VEL
LIN {X 0,Y 608.45,Z 508.689,A -85,B 0,C 180,E1 -530.023,E2 -530.023} C_VEL
LIN {X 0,Y 608.474,Z 508.685,A -85,B 0,C 180,E1 -532.701,E2 -532.701} C_VEL
LIN {X 0,Y 608.464,Z 508.695,A -85,B 0,C 180,E1 -535.362,E2 -535.362} C_VEL
LIN {X 0,Y 608.446,Z 508.69,A -85,B 0,C 180,E1 -538.014,E2 -538.014} C_VEL
LIN {X 0,Y 608.478,Z 508.684,A -85,B 0,C 180,E1 -540.662,E2 -540.662} C_VEL
LIN {X 0,Y 608.478,Z 508.693,A -85,B 0,C 180,E1 -543.311,E2 -543.311} C_VEL
LIN {X 0,Y 608.453,Z 508.689,A -85,B 0,C 180,E1 -545.967,E2 -545.967} C_VEL
LIN {X 0,Y 608.457,Z 508.687,A -85,B 0,C 180,E1 -548.636,E2 -548.636} C_VEL
LIN {X 0,Y 608.452,Z 508.693,A -85,B 0,C 180,E1 -549.471,E2 -549.471} C_VEL
LIN {X 0,Y 607.772,Z 508.774,A -85,B 0,C 180,E1 -550.024,E2 -550.024} C_VEL
LIN {X 0,Y 604.917,Z 509.13,A -85,B 0,C 180,E1 -550.921,E2 -550.921} C_VEL
LIN {X 0,Y 602.516,Z 509.434,A -85,B 0,C 180,E1 -551.642,E2 -551.642} C_VEL
LIN {X 0,Y 601.488,Z 509.556,A -85,B 0,C 180,E1 -552.199,E2 -552.199} C_VEL
LIN {X 0,Y 601.406,Z 509.565,A -85,B 0,C 180,E1 -552.388,E2 -552.388} C_VEL
LIN {X 0,Y 601.426,Z 509.565,A -85,B 0,C 180,E1 -554.897,E2 -554.897} C_VEL
LIN {X 0,Y 601.426,Z 509.566,A -85,B 0,C 180,E1 -556.986,E2 -556.986} C_VEL
LIN {X 0,Y 601.402,Z 509.57,A -85,B 0,C 180,E1 -559.81,E2 -559.81} C_VEL
LIN {X 0,Y 601.406,Z 509.565,A -85,B 0,C 180,E1 -562.606,E2 -562.606} C_VEL
LIN {X 0,Y 601.399,Z 509.568,A -85,B 0,C 180,E1 -564.879,E2 -564.879} C_VEL
LIN {X 0,Y 601.417,Z 509.567,A -85,B 0,C 180,E1 -567.868,E2 -567.868} C_VEL
LIN {X 0,Y 601.441,Z 509.561,A -85,B 0,C 180,E1 -570.164,E2 -570.164} C_VEL
LIN {X 0,Y 601.418,Z 509.564,A -85,B 0,C 180,E1 -572.717,E2 -572.717} C_VEL
LIN {X 0,Y 601.417,Z 509.569,A -85,B 0,C 180,E1 -575.117,E2 -575.117} C_VEL
LIN {X 0,Y 601.43,Z 509.573,A -85,B 0,C 180,E1 -577.42,E2 -577.42} C_VEL
LIN {X 0,Y 601.407,Z 509.567,A -85,B 0,C 180,E1 -579.996,E2 -579.996} C_VEL
LIN {X 0,Y 601.406,Z 509.566,A -85,B 0,C 180,E1 -582.671,E2 -582.671} C_VEL
LIN {X 0,Y 601.422,Z 509.572,A -85,B 0,C 180,E1 -585.483,E2 -585.483} C_VEL
LIN {X 0,Y 601.423,Z 509.563,A -85,B 0,C 180,E1 -588.408,E2 -588.408} C_VEL
LIN {X 0,Y 601.433,Z 509.564,A -85,B 0,C 180,E1 -590.876,E2 -590.876} C_VEL
LIN {X 0,Y 601.432,Z 509.567,A -85,B 0,C 180,E1 -593.736,E2 -593.736} C_VEL
LIN {X 0,Y 601.42,Z 509.564,A -85,B 0,C 180,E1 -596.687,E2 -596.687} C_VEL
LIN {X 0,Y 601.424,Z 509.568,A -85,B 0,C 180,E1 -599.059,E2 -599.059} C_VEL
LIN {X 0,Y 601.434,Z 509.572,A -85,B 0,C 180,E1 -601.374,E2 -601.374} C_VEL
LIN {X 0,Y 601.405,Z 509.571,A -85,B 0,C 180,E1 -603.637,E2 -603.637} C_VEL
LIN {X 0,Y 601.462,Z 509.561,A -85,B 0,C 180,E1 -605.86,E2 -605.86} C_VEL
LIN {X 0,Y 601.406,Z 509.567,A -85,B 0,C 180,E1 -608.761,E2 -608.761} C_VEL
LIN {X 0,Y 601.425,Z 509.57,A -85,B 0,C 180,E1 -611.609,E2 -611.609} C_VEL
LIN {X 0,Y 601.417,Z 509.565,A -85,B 0,C 180,E1 -614.409,E2 -614.409} C_VEL
LIN {X 0,Y 601.438,Z 509.578,A -85,B 0,C 180,E1 -614.627,E2 -614.627} C_VEL
LIN {X 0,Y 601.469,Z 523.7,A -85,B 0,C 180,E1 -617.002,E2 -617.002} C_VEL
LIN {X 0,Y 601.435,Z 541.224,A -85,B 0,C 180,E1 -619.905,E2 -619.905} C_VEL
LIN {X 0,Y 601.426,Z 547.166,A -85,B 0,C 180,E1 -620.881,E2 -620.881} C_VEL
LIN {X 0,Y 601.688,Z 557.226,A -85,B 0,C 180,E1 -621.012,E2 -621.012} C_VEL
LIN {X 0,Y 601.583,Z 654.525,A -85,B 0,C 180,E1 -622.195,E2 -622.195} C_VEL
LIN {X 0,Y 601.568,Z 668.227,A -85,B 0,C 180,E1 -622.511,E2 -622.511} C_VEL
LIN {X 0,Y 601.54,Z 680.756,A -85,B 0,C 180,E1 -622.941,E2 -622.941} C_VEL
LIN {X 0,Y 601.492,Z 692.688,A -85,B 0,C 180,E1 -623.497,E2 -623.497} C_VEL
LIN {X 0,Y 601.468,Z 704.634,A -85,B 0,C 180,E1 -624.216,E2 -624.216} C_VEL
LIN {X 0,Y 601.456,Z 714.689,A -85,B 0,C 180,E1 -624.972,E2 -624.972} C_VEL
LIN {X 0,Y 601.414,Z 723.758,A -85,B 0,C 180,E1 -625.812,E2 -625.812} C_VEL
LIN {X 0,Y 601.392,Z 732.61,A -85,B 0,C 180,E1 -626.818,E2 -626.818} C_VEL
LIN {X 0,Y 601.385,Z 739.748,A -85,B 0,C 180,E1 -627.823,E2 -627.823} C_VEL
LIN {X 0,Y 601.381,Z 746.264,A -85,B 0,C 180,E1 -628.996,E2 -628.996} C_VEL
LIN {X 0,Y 601.358,Z 750.588,A -85,B 0,C 180,E1 -630,E2 -630} C_VEL
LIN {X 0,Y 601.34,Z 752.876,A -85,B 0,C 180,E1 -630.67,E2 -630.67} C_VEL
LIN {X 0,Y 601.348,Z 754.742,A -85,B 0,C 180,E1 -631.339,E2 -631.339} C_VEL
LIN {X 0,Y 601.343,Z 756.158,A -85,B 0,C 180,E1 -632.009,E2 -632.009} C_VEL
LIN {X 0,Y 601.338,Z 757.766,A -85,B 0,C 180,E1 -633.35,E2 -633.35} C_VEL
LIN {X 0,Y 601.342,Z 757.999,A -85,B 0,C 180,E1 -634.021,E2 -634.021} C_VEL
LIN {X 0,Y 601.337,Z 757.207,A -85,B 0,C 180,E1 -635.365,E2 -635.365} C_VEL
LIN {X 0,Y 601.363,Z 755.101,A -85,B 0,C 180,E1 -636.595,E2 -636.595} C_VEL
LIN {X 0,Y 601.34,Z 751.917,A -85,B 0,C 180,E1 -637.724,E2 -637.724} C_VEL
LIN {X 0,Y 601.35,Z 747.945,A -85,B 0,C 180,E1 -638.739,E2 -638.739} C_VEL
LIN {X 0,Y 601.362,Z 741.807,A -85,B 0,C 180,E1 -639.926,E2 -639.926} C_VEL
LIN {X 0,Y 601.387,Z 734.75,A -85,B 0,C 180,E1 -640.991,E2 -640.991} C_VEL
LIN {X 0,Y 601.431,Z 726.69,A -85,B 0,C 180,E1 -641.971,E2 -641.971} C_VEL
LIN {X 0,Y 601.426,Z 718.023,A -85,B 0,C 180,E1 -642.828,E2 -642.828} C_VEL
LIN {X 0,Y 601.48,Z 707.814,A -85,B 0,C 180,E1 -643.65,E2 -643.65} C_VEL
LIN {X 0,Y 601.506,Z 696.64,A -85,B 0,C 180,E1 -644.376,E2 -644.376} C_VEL
LIN {X 0,Y 601.541,Z 684.687,A -85,B 0,C 180,E1 -644.98,E2 -644.98} C_VEL
LIN {X 0,Y 601.554,Z 672.213,A -85,B 0,C 180,E1 -645.457,E2 -645.457} C_VEL
LIN {X 0,Y 601.59,Z 659.331,A -85,B 0,C 180,E1 -645.803,E2 -645.803} C_VEL
LIN {X 0,Y 601.592,Z 645.627,A -85,B 0,C 180,E1 -646.021,E2 -646.021} C_VEL
LIN {X 0,Y 601.503,Z 547.764,A -85,B 0,C 180,E1 -647.195,E2 -647.195} C_VEL
LIN {X 0,Y 601.427,Z 547.192,A -85,B 0,C 180,E1 -647.204,E2 -647.204} C_VEL
LIN {X 0,Y 601.486,Z 529.258,A -85,B 0,C 180,E1 -650.162,E2 -650.162} C_VEL
LIN {X 0,Y 601.535,Z 512.058,A -85,B 0,C 180,E1 -653.041,E2 -653.041} C_VEL
LIN {X 0,Y 601.434,Z 509.564,A -85,B 0,C 180,E1 -653.5,E2 -653.5} C_VEL
LIN {X 0,Y 601.404,Z 509.571,A -85,B 0,C 180,E1 -656.363,E2 -656.363} C_VEL
LIN {X 0,Y 601.44,Z 509.57,A -85,B 0,C 180,E1 -658.789,E2 -658.789} C_VEL
LIN {X 0,Y 601.43,Z 509.563,A -85,B 0,C 180,E1 -661.456,E2 -661.456} C_VEL
LIN {X 0,Y 601.43,Z 509.564,A -85,B 0,C 180,E1 -664.117,E2 -664.117} C_VEL
LIN {X 0,Y 601.414,Z 509.573,A -85,B 0,C 180,E1 -666.581,E2 -666.581} C_VEL
LIN {X 0,Y 601.436,Z 509.561,A -85,B 0,C 180,E1 -669.535,E2 -669.535} C_VEL
LIN {X 0,Y 601.435,Z 509.572,A -85,B 0,C 180,E1 -672.667,E2 -672.667} C_VEL
LIN {X 0,Y 601.422,Z 509.563,A -85,B 0,C 180,E1 -675.481,E2 -675.481} C_VEL
LIN {X 0,Y 601.424,Z 509.569,A -85,B 0,C 180,E1 -678.405,E2 -678.405} C_VEL
LIN {X 0,Y 601.432,Z 509.569,A -85,B 0,C 180,E1 -680.875,E2 -680.875} C_VEL
LIN {X 0,Y 601.438,Z 509.561,A -85,B 0,C 180,E1 -683.733,E2 -683.733} C_VEL
LIN {X 0,Y 601.433,Z 509.563,A -85,B 0,C 180,E1 -686.062,E2 -686.062} C_VEL
LIN {X 0,Y 601.436,Z 509.57,A -85,B 0,C 180,E1 -688.541,E2 -688.541} C_VEL
LIN {X 0,Y 601.43,Z 509.563,A -85,B 0,C 180,E1 -691.373,E2 -691.373} C_VEL
LIN {X 0,Y 601.416,Z 509.566,A -85,B 0,C 180,E1 -694.129,E2 -694.129} C_VEL
LIN {X 0,Y 601.418,Z 509.573,A -85,B 0,C 180,E1 -696.589,E2 -696.589} C_VEL
LIN {X 0,Y 601.427,Z 509.563,A -85,B 0,C 180,E1 -699.478,E2 -699.478} C_VEL
LIN {X 0,Y 601.395,Z 509.571,A -85,B 0,C 180,E1 -702.311,E2 -702.311} C_VEL
LIN {X 0,Y 601.41,Z 509.571,A -85,B 0,C 180,E1 -704.408,E2 -704.408} C_VEL
LIN {X 0,Y 601.419,Z 509.565,A -85,B 0,C 180,E1 -707.172,E2 -707.172} C_VEL
LIN {X 0,Y 601.428,Z 509.563,A -85,B 0,C 180,E1 -709.905,E2 -709.905} C_VEL
LIN {X 0,Y 601.447,Z 509.571,A -85,B 0,C 180,E1 -712.615,E2 -712.615} C_VEL
LIN {X 0,Y 601.429,Z 509.563,A -85,B 0,C 180,E1 -715.308,E2 -715.308} C_VEL
LIN {X 0,Y 601.418,Z 509.565,A -85,B 0,C 180,E1 -717.991,E2 -717.991} C_VEL
LIN {X 0,Y 601.448,Z 509.57,A -85,B 0,C 180,E1 -720.669,E2 -720.669} C_VEL
LIN {X 0,Y 601.427,Z 509.563,A -85,B 0,C 180,E1 -723.35,E2 -723.35} C_VEL
LIN {X 0,Y 601.406,Z 509.567,A -85,B 0,C 180,E1 -726.037,E2 -726.037} C_VEL
LIN {X 0,Y 601.436,Z 509.569,A -85,B 0,C 180,E1 -728.738,E2 -728.738} C_VEL
LIN {X 0,Y 601.426,Z 509.563,A -85,B 0,C 180,E1 -731.458,E2 -731.458} C_VEL
LIN {X 0,Y 601.409,Z 509.568,A -85,B 0,C 180,E1 -734.206,E2 -734.206} C_VEL
LIN {X 0,Y 601.426,Z 509.566,A -85,B 0,C 180,E1 -736.986,E2 -736.986} C_VEL
LIN {X 0,Y 601.4,Z 509.566,A -85,B 0,C 180,E1 -739.81,E2 -739.81} C_VEL
LIN {X 0,Y 601.406,Z 509.576,A -85,B 0,C 180,E1 -742.606,E2 -742.606} C_VEL
LIN {X 0,Y 601.398,Z 509.571,A -85,B 0,C 180,E1 -744.879,E2 -744.879} C_VEL
LIN {X 0,Y 601.415,Z 509.564,A -85,B 0,C 180,E1 -747.868,E2 -747.868} C_VEL
LIN {X 0,Y 601.44,Z 509.565,A -85,B 0,C 180,E1 -750.163,E2 -750.163} C_VEL
LIN {X 0,Y 601.419,Z 509.572,A -85,B 0,C 180,E1 -752.717,E2 -752.717} C_VEL
LIN {X 0,Y 601.415,Z 509.566,A -85,B 0,C 180,E1 -755.116,E2 -755.116} C_VEL
LIN {X 0,Y 601.428,Z 509.562,A -85,B 0,C 180,E1 -757.42,E2 -757.42} C_VEL
LIN {X 0,Y 601.409,Z 509.567,A -85,B 0,C 180,E1 -759.995,E2 -759.995} C_VEL
LIN {X 0,Y 601.405,Z 509.574,A -85,B 0,C 180,E1 -762.671,E2 -762.671} C_VEL
LIN {X 0,Y 601.421,Z 509.563,A -85,B 0,C 180,E1 -765.483,E2 -765.483} C_VEL
LIN {X 0,Y 601.427,Z 509.571,A -85,B 0,C 180,E1 -768.407,E2 -768.407} C_VEL
LIN {X 0,Y 601.433,Z 509.567,A -85,B 0,C 180,E1 -770.876,E2 -770.876} C_VEL
LIN {X 0,Y 601.405,Z 509.566,A -85,B 0,C 180,E1 -773.739,E2 -773.739} C_VEL
LIN {X 0,Y 601.429,Z 509.57,A -85,B 0,C 180,E1 -776.687,E2 -776.687} C_VEL
LIN {X 0,Y 601.431,Z 509.564,A -85,B 0,C 180,E1 -779.06,E2 -779.06} C_VEL
LIN {X 0,Y 601.427,Z 509.563,A -85,B 0,C 180,E1 -781.374,E2 -781.374} C_VEL
LIN {X 0,Y 601.4,Z 509.566,A -85,B 0,C 180,E1 -783.637,E2 -783.637} C_VEL
LIN {X 0,Y 601.42,Z 509.574,A -85,B 0,C 180,E1 -786.59,E2 -786.59} C_VEL
LIN {X 0,Y 601.467,Z 509.766,A -85,B 0,C 180,E1 -787.581,E2 -787.581} C_VEL
LIN {X 0,Y 601.611,Z 520.752,A -85,B 0,C 180,E1 -789.157,E2 -789.157} C_VEL
LIN {X 0,Y 601.558,Z 540.692,A -85,B 0,C 180,E1 -791.965,E2 -791.965} C_VEL
LIN {X 0,Y 601.492,Z 560.841,A -85,B 0,C 180,E1 -794.758,E2 -794.758} C_VEL
LIN {X 0,Y 601.466,Z 576.169,A -85,B 0,C 180,E1 -796.83,E2 -796.83} C_VEL
LIN {X 0,Y 601.639,Z 594.056,A -85,B 0,C 180,E1 -797.048,E2 -797.048} C_VEL
LIN {X 0,Y 601.603,Z 683.962,A -85,B 0,C 180,E1 -798.14,E2 -798.14} C_VEL
LIN {X 0,Y 601.579,Z 697.227,A -85,B 0,C 180,E1 -798.438,E2 -798.438} C_VEL
LIN {X 0,Y 601.547,Z 708.926,A -85,B 0,C 180,E1 -798.826,E2 -798.826} C_VEL
LIN {X 0,Y 601.515,Z 719.928,A -85,B 0,C 180,E1 -799.311,E2 -799.311} C_VEL
LIN {X 0,Y 601.466,Z 730.584,A -85,B 0,C 180,E1 -799.906,E2 -799.906} C_VEL
LIN {X 0,Y 601.445,Z 741.478,A -85,B 0,C 180,E1 -800.67,E2 -800.67} C_VEL
LIN {X 0,Y 601.429,Z 752.114,A -85,B 0,C 180,E1 -801.601,E2 -801.601} C_VEL
LIN {X 0,Y 601.418,Z 759.962,A -85,B 0,C 180,E1 -802.446,E2 -802.446} C_VEL
LIN {X 0,Y 601.37,Z 767.225,A -85,B 0,C 180,E1 -803.398,E2 -803.398} C_VEL
LIN {X 0,Y 601.371,Z 772.867,A -85,B 0,C 180,E1 -804.299,E2 -804.299} C_VEL
LIN {X 0,Y 601.337,Z 777.951,A -85,B 0,C 180,E1 -805.307,E2 -805.307} C_VEL
LIN {X 0,Y 601.367,Z 781.896,A -85,B 0,C 180,E1 -806.315,E2 -806.315} C_VEL
LIN {X 0,Y 601.325,Z 784.809,A -85,B 0,C 180,E1 -807.321,E2 -807.321} C_VEL
LIN {X 0,Y 601.34,Z 786.202,A -85,B 0,C 180,E1 -807.991,E2 -807.991} C_VEL
LIN {X 0,Y 601.339,Z 787.784,A -85,B 0,C 180,E1 -809.33,E2 -809.33} C_VEL
LIN {X 0,Y 601.335,Z 788,A -85,B 0,C 180,E1 -810,E2 -810} C_VEL
LIN {X 0,Y 601.348,Z 787.184,A -85,B 0,C 180,E1 -811.339,E2 -811.339} C_VEL
LIN {X 0,Y 601.34,Z 786.202,A -85,B 0,C 180,E1 -812.009,E2 -812.009} C_VEL
LIN {X 0,Y 601.325,Z 784.809,A -85,B 0,C 180,E1 -812.679,E2 -812.679} C_VEL
LIN {X 0,Y 601.367,Z 781.896,A -85,B 0,C 180,E1 -813.685,E2 -813.685} C_VEL
LIN {X 0,Y 601.337,Z 777.95,A -85,B 0,C 180,E1 -814.693,E2 -814.693} C_VEL
LIN {X 0,Y 601.372,Z 771.878,A -85,B 0,C 180,E1 -815.869,E2 -815.869} C_VEL
LIN {X 0,Y 601.382,Z 765.237,A -85,B 0,C 180,E1 -816.88,E2 -816.88} C_VEL
LIN {X 0,Y 601.4,Z 756.991,A -85,B 0,C 180,E1 -817.892,E2 -817.892} C_VEL
LIN {X 0,Y 601.436,Z 748.539,A -85,B 0,C 180,E1 -818.737,E2 -818.737} C_VEL
LIN {X 0,Y 601.442,Z 738.095,A -85,B 0,C 180,E1 -819.585,E2 -819.585} C_VEL
LIN {X 0,Y 601.484,Z 727.761,A -85,B 0,C 180,E1 -820.264,E2 -820.264} C_VEL
LIN {X 0,Y 601.537,Z 716.901,A -85,B 0,C 180,E1 -820.836,E2 -820.836} C_VEL
LIN {X 0,Y 601.559,Z 704.381,A -85,B 0,C 180,E1 -821.34,E2 -821.34} C_VEL
LIN {X 0,Y 601.59,Z 691.364,A -85,B 0,C 180,E1 -821.711,E2 -821.711} C_VEL
LIN {X 0,Y 601.61,Z 678.106,A -85,B 0,C 180,E1 -821.946,E2 -821.946} C_VEL
LIN {X 0,Y 601.568,Z 576.839,A -85,B 0,C 180,E1 -823.16,E2 -823.16} C_VEL
LIN {X 0,Y 601.471,Z 575.637,A -85,B 0,C 180,E1 -823.213,E2 -823.213} C_VEL
LIN {X 0,Y 601.495,Z 554.544,A -85,B 0,C 180,E1 -826.111,E2 -826.111} C_VEL
LIN {X 0,Y 601.561,Z 536.5,A -85,B 0,C 180,E1 -828.621,E2 -828.621} C_VEL
LIN {X 0,Y 601.659,Z 515.506,A -85,B 0,C 180,E1 -831.589,E2 -831.589} C_VEL
LIN {X 0,Y 601.419,Z 509.567,A -85,B 0,C 180,E1 -832.461,E2 -832.461} C_VEL
LIN {X 0,Y 601.403,Z 509.568,A -85,B 0,C 180,E1 -834.878,E2 -834.878} C_VEL
LIN {X 0,Y 601.42,Z 509.568,A -85,B 0,C 180,E1 -837.867,E2 -837.867} C_VEL
LIN {X 0,Y 601.428,Z 509.563,A -85,B 0,C 180,E1 -840.163,E2 -840.163} C_VEL
LIN {X 0,Y 601.42,Z 509.564,A -85,B 0,C 180,E1 -842.715,E2 -842.715} C_VEL
LIN {X 0,Y 601.392,Z 509.571,A -85,B 0,C 180,E1 -845.111,E2 -845.111} C_VEL
LIN {X 0,Y 601.435,Z 509.571,A -85,B 0,C 180,E1 -847.418,E2 -847.418} C_VEL
LIN {X 0,Y 601.409,Z 509.567,A -85,B 0,C 180,E1 -849.994,E2 -849.994} C_VEL
LIN {X 0,Y 601.411,Z 509.565,A -85,B 0,C 180,E1 -852.669,E2 -852.669} C_VEL
LIN {X 0,Y 601.421,Z 509.574,A -85,B 0,C 180,E1 -855.481,E2 -855.481} C_VEL
LIN {X 0,Y 601.418,Z 509.563,A -85,B 0,C 180,E1 -858.406,E2 -858.406} C_VEL
LIN {X 0,Y 601.431,Z 509.564,A -85,B 0,C 180,E1 -860.875,E2 -860.875} C_VEL
LIN {X 0,Y 601.438,Z 509.567,A -85,B 0,C 180,E1 -863.733,E2 -863.733} C_VEL
LIN {X 0,Y 601.43,Z 509.564,A -85,B 0,C 180,E1 -866.063,E2 -866.063} C_VEL
LIN {X 0,Y 601.434,Z 509.561,A -85,B 0,C 180,E1 -868.541,E2 -868.541} C_VEL
LIN {X 0,Y 601.43,Z 509.571,A -85,B 0,C 180,E1 -871.373,E2 -871.373} C_VEL
LIN {X 0,Y 601.415,Z 509.565,A -85,B 0,C 180,E1 -874.129,E2 -874.129} C_VEL
LIN {X 0,Y 601.416,Z 509.564,A -85,B 0,C 180,E1 -876.589,E2 -876.589} C_VEL
LIN {X 0,Y 601.427,Z 509.573,A -85,B 0,C 180,E1 -879.478,E2 -879.478} C_VEL
LIN {X 0,Y 601.392,Z 509.567,A -85,B 0,C 180,E1 -882.311,E2 -882.311} C_VEL
LIN {X 0,Y 601.408,Z 509.565,A -85,B 0,C 180,E1 -884.409,E2 -884.409} C_VEL
LIN {X 0,Y 601.417,Z 509.569,A -85,B 0,C 180,E1 -887.172,E2 -887.172} C_VEL
LIN {X 0,Y 601.428,Z 509.565,A -85,B 0,C 180,E1 -889.905,E2 -889.905} C_VEL
LIN {X 0,Y 601.444,Z 509.56,A -85,B 0,C 180,E1 -892.615,E2 -892.615} C_VEL
LIN {X 0,Y 601.43,Z 509.57,A -85,B 0,C 180,E1 -895.308,E2 -895.308} C_VEL
LIN {X 0,Y 601.416,Z 509.566,A -85,B 0,C 180,E1 -897.991,E2 -897.991} C_VEL
LIN {X 0,Y 601.448,Z 509.56,A -85,B 0,C 180,E1 -900.67,E2 -900.67} C_VEL
LIN {X 0,Y 601.429,Z 509.572,A -85,B 0,C 180,E1 -903.35,E2 -903.35} C_VEL
LIN {X 0,Y 601.406,Z 509.567,A -85,B 0,C 180,E1 -906.037,E2 -906.037} C_VEL
LIN {X 0,Y 601.435,Z 509.562,A -85,B 0,C 180,E1 -908.738,E2 -908.738} C_VEL
LIN {X 0,Y 601.427,Z 509.573,A -85,B 0,C 180,E1 -911.458,E2 -911.458} C_VEL
LIN {X 0,Y 601.406,Z 509.565,A -85,B 0,C 180,E1 -912.388,E2 -912.388} C_VEL
LIN {X 0,Y 600.743,Z 509.652,A -85,B 0,C 180,E1 -912.947,E2 -912.947} C_VEL
LIN {X 0,Y 597.892,Z 510.006,A -85,B 0,C 180,E1 -913.855,E2 -913.855} C_VEL
LIN {X 0,Y 595.48,Z 510.307,A -85,B 0,C 180,E1 -914.585,E2 -914.585} C_VEL
LIN {X 0,Y 594.442,Z 510.438,A -85,B 0,C 180,E1 -915.148,E2 -915.148} C_VEL
LIN {X 0,Y 594.357,Z 510.446,A -85,B 0,C 180,E1 -915.339,E2 -915.339} C_VEL
LIN {X 0,Y 594.373,Z 510.444,A -85,B 0,C 180,E1 -917.905,E2 -917.905} C_VEL
LIN {X 0,Y 594.377,Z 510.443,A -85,B 0,C 180,E1 -920.919,E2 -920.919} C_VEL
LIN {X 0,Y 594.385,Z 510.445,A -85,B 0,C 180,E1 -923.704,E2 -923.704} C_VEL
LIN {X 0,Y 594.382,Z 510.441,A -85,B 0,C 180,E1 -926.7,E2 -926.7} C_VEL
LIN {X 0,Y 594.379,Z 510.444,A -85,B 0,C 180,E1 -928.999,E2 -928.999} C_VEL
LIN {X 0,Y 594.387,Z 510.446,A -85,B 0,C 180,E1 -931.646,E2 -931.646} C_VEL
LIN {X 0,Y 594.394,Z 510.439,A -85,B 0,C 180,E1 -934.579,E2 -934.579} C_VEL
LIN {X 0,Y 594.38,Z 510.445,A -85,B 0,C 180,E1 -937.087,E2 -937.087} C_VEL
LIN {X 0,Y 594.373,Z 510.445,A -85,B 0,C 180,E1 -939.776,E2 -939.776} C_VEL
LIN {X 0,Y 594.364,Z 510.442,A -85,B 0,C 180,E1 -942.376,E2 -942.376} C_VEL
LIN {X 0,Y 594.36,Z 510.45,A -85,B 0,C 180,E1 -945.192,E2 -945.192} C_VEL
LIN {X 0,Y 594.385,Z 510.446,A -85,B 0,C 180,E1 -947.627,E2 -947.627} C_VEL
LIN {X 0,Y 594.389,Z 510.439,A -85,B 0,C 180,E1 -950.322,E2 -950.322} C_VEL
LIN {X 0,Y 594.385,Z 510.442,A -85,B 0,C 180,E1 -952.914,E2 -952.914} C_VEL
LIN {X 0,Y 594.382,Z 510.443,A -85,B 0,C 180,E1 -955.862,E2 -955.862} C_VEL
LIN {X 0,Y 594.38,Z 510.441,A -85,B 0,C 180,E1 -958.651,E2 -958.651} C_VEL
LIN {X 0,Y 594.384,Z 510.444,A -85,B 0,C 180,E1 -961.043,E2 -961.043} C_VEL
LIN {X 0,Y 594.384,Z 510.442,A -85,B 0,C 180,E1 -963.979,E2 -963.979} C_VEL
LIN {X 0,Y 594.38,Z 510.44,A -85,B 0,C 180,E1 -966.296,E2 -966.296} C_VEL
LIN {X 0,Y 594.406,Z 510.445,A -85,B 0,C 180,E1 -969.225,E2 -969.225} C_VEL
LIN {X 0,Y 594.356,Z 510.445,A -85,B 0,C 180,E1 -972.096,E2 -972.096} C_VEL
LIN {X 0,Y 594.433,Z 510.525,A -85,B 0,C 180,E1 -974.551,E2 -974.551} C_VEL
LIN {X 0,Y 594.472,Z 522.974,A -85,B 0,C 180,E1 -976.672,E2 -976.672} C_VEL
LIN {X 0,Y 594.42,Z 539.46,A -85,B 0,C 180,E1 -979.441,E2 -979.441} C_VEL
LIN {X 0,Y 594.395,Z 547.358,A -85,B 0,C 180,E1 -980.73,E2 -980.73} C_VEL
LIN {X 0,Y 594.767,Z 552.433,A -85,B 0,C 180,E1 -980.8,E2 -980.8} C_VEL
LIN {X 0,Y 594.647,Z 653.702,A -85,B 0,C 180,E1 -982.039,E2 -982.039} C_VEL
LIN {X 0,Y 594.626,Z 666.933,A -85,B 0,C 180,E1 -982.338,E2 -982.338} C_VEL
LIN {X 0,Y 594.576,Z 679.59,A -85,B 0,C 180,E1 -982.764,E2 -982.764} C_VEL
LIN {X 0,Y 594.519,Z 691.288,A -85,B 0,C 180,E1 -983.296,E2 -983.296} C_VEL
LIN {X 0,Y 594.472,Z 702.827,A -85,B 0,C 180,E1 -983.977,E2 -983.977} C_VEL
LIN {X 0,Y 594.42,Z 713.201,A -85,B 0,C 180,E1 -984.743,E2 -984.743} C_VEL
LIN {X 0,Y 594.372,Z 722.592,A -85,B 0,C 180,E1 -985.592,E2 -985.592} C_VEL
LIN {X 0,Y 594.298,Z 731.648,A -85,B 0,C 180,E1 -986.61,E2 -986.61} C_VEL
LIN {X 0,Y 594.329,Z 738.957,A -85,B 0,C 180,E1 -987.628,E2 -987.628} C_VEL
LIN {X 0,Y 594.264,Z 744.833,A -85,B 0,C 180,E1 -988.645,E2 -988.645} C_VEL
LIN {X 0,Y 594.299,Z 749.474,A -85,B 0,C 180,E1 -989.661,E2 -989.661} C_VEL
LIN {X 0,Y 594.241,Z 753.028,A -85,B 0,C 180,E1 -990.678,E2 -990.678} C_VEL
LIN {X 0,Y 594.248,Z 754.862,A -85,B 0,C 180,E1 -991.355,E2 -991.355} C_VEL
LIN {X 0,Y 594.242,Z 756.237,A -85,B 0,C 180,E1 -992.033,E2 -992.033} C_VEL
LIN {X 0,Y 594.258,Z 757.8,A -85,B 0,C 180,E1 -993.39,E2 -993.39} C_VEL
LIN {X 0,Y 594.255,Z 757.999,A -85,B 0,C 180,E1 -994.069,E2 -994.069} C_VEL
LIN {X 0,Y 594.252,Z 757.152,A -85,B 0,C 180,E1 -995.429,E2 -995.429} C_VEL
LIN {X 0,Y 594.261,Z 755.213,A -85,B 0,C 180,E1 -996.572,E2 -996.572} C_VEL
LIN {X 0,Y 594.245,Z 751.755,A -85,B 0,C 180,E1 -997.817,E2 -997.817} C_VEL
LIN {X 0,Y 594.253,Z 747.733,A -85,B 0,C 180,E1 -998.844,E2 -998.844} C_VEL
LIN {X 0,Y 594.287,Z 741.515,A -85,B 0,C 180,E1 -1000.045,E2 -1000.045} C_VEL
LIN {X 0,Y 594.315,Z 735.038,A -85,B 0,C 180,E1 -1001.034,E2 -1001.034} C_VEL
LIN {X 0,Y 594.381,Z 726.241,A -85,B 0,C 180,E1 -1002.115,E2 -1002.115} C_VEL
LIN {X 0,Y 594.386,Z 717.462,A -85,B 0,C 180,E1 -1002.982,E2 -1002.982} C_VEL
LIN {X 0,Y 594.436,Z 707.391,A -85,B 0,C 180,E1 -1003.796,E2 -1003.796} C_VEL
LIN {X 0,Y 594.498,Z 697.258,A -85,B 0,C 180,E1 -1004.461,E2 -1004.461} C_VEL
LIN {X 0,Y 594.566,Z 685.548,A -85,B 0,C 180,E1 -1005.073,E2 -1005.073} C_VEL
LIN {X 0,Y 594.611,Z 673.349,A -85,B 0,C 180,E1 -1005.554,E2 -1005.554} C_VEL
LIN {X 0,Y 594.642,Z 660.006,A -85,B 0,C 180,E1 -1005.927,E2 -1005.927} C_VEL
LIN {X 0,Y 594.667,Z 646.948,A -85,B 0,C 180,E1 -1006.146,E2 -1006.146} C_VEL
LIN {X 0,Y 594.589,Z 548.411,A -85,B 0,C 180,E1 -1007.343,E2 -1007.343} C_VEL
LIN {X 0,Y 594.407,Z 547.15,A -85,B 0,C 180,E1 -1007.37,E2 -1007.37} C_VEL
LIN {X 0,Y 594.449,Z 528.942,A -85,B 0,C 180,E1 -1010.412,E2 -1010.412} C_VEL
LIN {X 0,Y 594.539,Z 511.738,A -85,B 0,C 180,E1 -1013.328,E2 -1013.328} C_VEL
LIN {X 0,Y 594.419,Z 510.439,A -85,B 0,C 180,E1 -1013.564,E2 -1013.564} C_VEL
LIN {X 0,Y 594.387,Z 510.45,A -85,B 0,C 180,E1 -1016.699,E2 -1016.699} C_VEL
LIN {X 0,Y 594.382,Z 510.446,A -85,B 0,C 180,E1 -1018.998,E2 -1018.998} C_VEL
LIN {X 0,Y 594.385,Z 510.44,A -85,B 0,C 180,E1 -1021.643,E2 -1021.643} C_VEL
LIN {X 0,Y 594.383,Z 510.449,A -85,B 0,C 180,E1 -1024.579,E2 -1024.579} C_VEL
LIN {X 0,Y 594.386,Z 510.443,A -85,B 0,C 180,E1 -1027.086,E2 -1027.086} C_VEL
LIN {X 0,Y 594.373,Z 510.441,A -85,B 0,C 180,E1 -1029.774,E2 -1029.774} C_VEL
LIN {X 0,Y 594.385,Z 510.445,A -85,B 0,C 180,E1 -1032.373,E2 -1032.373} C_VEL
LIN {X 0,Y 594.36,Z 510.445,A -85,B 0,C 180,E1 -1035.19,E2 -1035.19} C_VEL
LIN {X 0,Y 594.364,Z 510.442,A -85,B 0,C 180,E1 -1037.624,E2 -1037.624} C_VEL
LIN {X 0,Y 594.389,Z 510.443,A -85,B 0,C 180,E1 -1040.32,E2 -1040.32} C_VEL
LIN {X 0,Y 594.38,Z 510.446,A -85,B 0,C 180,E1 -1042.913,E2 -1042.913} C_VEL
LIN {X 0,Y 594.383,Z 510.44,A -85,B 0,C 180,E1 -1045.859,E2 -1045.859} C_VEL
LIN {X 0,Y 594.385,Z 510.451,A -85,B 0,C 180,E1 -1048.65,E2 -1048.65} C_VEL
LIN {X 0,Y 594.381,Z 510.444,A -85,B 0,C 180,E1 -1051.04,E2 -1051.04} C_VEL
LIN {X 0,Y 594.388,Z 510.44,A -85,B 0,C 180,E1 -1053.974,E2 -1053.974} C_VEL
LIN {X 0,Y 594.385,Z 510.444,A -85,B 0,C 180,E1 -1056.296,E2 -1056.296} C_VEL
LIN {X 0,Y 594.401,Z 510.44,A -85,B 0,C 180,E1 -1059.224,E2 -1059.224} C_VEL
LIN {X 0,Y 594.375,Z 510.443,A -85,B 0,C 180,E1 -1062.095,E2 -1062.095} C_VEL
LIN {X 0,Y 594.363,Z 510.446,A -85,B 0,C 180,E1 -1064.219,E2 -1064.219} C_VEL
LIN {X 0,Y 594.365,Z 510.446,A -85,B 0,C 180,E1 -1067.017,E2 -1067.017} C_VEL
LIN {X 0,Y 594.388,Z 510.439,A -85,B 0,C 180,E1 -1069.784,E2 -1069.784} C_VEL
LIN {X 0,Y 594.411,Z 510.445,A -85,B 0,C 180,E1 -1072.527,E2 -1072.527} C_VEL
LIN {X 0,Y 594.397,Z 510.44,A -85,B 0,C 180,E1 -1075.252,E2 -1075.252} C_VEL
LIN {X 0,Y 594.388,Z 510.44,A -85,B 0,C 180,E1 -1077.967,E2 -1077.967} C_VEL
LIN {X 0,Y 594.418,Z 510.445,A -85,B 0,C 180,E1 -1080.677,E2 -1080.677} C_VEL
LIN {X 0,Y 594.378,Z 510.44,A -85,B 0,C 180,E1 -1083.389,E2 -1083.389} C_VEL
LIN {X 0,Y 594.362,Z 510.445,A -85,B 0,C 180,E1 -1086.109,E2 -1086.109} C_VEL
LIN {X 0,Y 594.395,Z 510.444,A -85,B 0,C 180,E1 -1088.842,E2 -1088.842} C_VEL
LIN {X 0,Y 594.385,Z 510.439,A -85,B 0,C 180,E1 -1091.596,E2 -1091.596} C_VEL
LIN {X 0,Y 594.38,Z 510.447,A -85,B 0,C 180,E1 -1094.377,E2 -1094.377} C_VEL
LIN {X 0,Y 594.383,Z 510.441,A -85,B 0,C 180,E1 -1097.194,E2 -1097.194} C_VEL
LIN {X 0,Y 594.37,Z 510.444,A -85,B 0,C 180,E1 -1100.054,E2 -1100.054} C_VEL
LIN {X 0,Y 594.357,Z 510.447,A -85,B 0,C 180,E1 -1102.968,E2 -1102.968} C_VEL
LIN {X 0,Y 594.373,Z 510.443,A -85,B 0,C 180,E1 -1105.193,E2 -1105.193} C_VEL
LIN {X 0,Y 594.376,Z 510.44,A -85,B 0,C 180,E1 -1107.527,E2 -1107.527} C_VEL
LIN {X 0,Y 594.392,Z 510.445,A -85,B 0,C 180,E1 -1110.331,E2 -1110.331} C_VEL
LIN {X 0,Y 594.372,Z 510.445,A -85,B 0,C 180,E1 -1112.951,E2 -1112.951} C_VEL
LIN {X 0,Y 594.379,Z 510.441,A -85,B 0,C 180,E1 -1115.407,E2 -1115.407} C_VEL
LIN {X 0,Y 594.38,Z 510.442,A -85,B 0,C 180,E1 -1117.941,E2 -1117.941} C_VEL
LIN {X 0,Y 594.374,Z 510.447,A -85,B 0,C 180,E1 -1120.823,E2 -1120.823} C_VEL
LIN {X 0,Y 594.361,Z 510.443,A -85,B 0,C 180,E1 -1123.3,E2 -1123.3} C_VEL
LIN {X 0,Y 594.378,Z 510.445,A -85,B 0,C 180,E1 -1126.16,E2 -1126.16} C_VEL
LIN {X 0,Y 594.378,Z 510.442,A -85,B 0,C 180,E1 -1129.178,E2 -1129.178} C_VEL
LIN {X 0,Y 594.386,Z 510.443,A -85,B 0,C 180,E1 -1132.06,E2 -1132.06} C_VEL
LIN {X 0,Y 594.35,Z 510.452,A -85,B 0,C 180,E1 -1134.677,E2 -1134.677} C_VEL
LIN {X 0,Y 594.378,Z 510.443,A -85,B 0,C 180,E1 -1137.089,E2 -1137.089} C_VEL
LIN {X 0,Y 594.387,Z 510.44,A -85,B 0,C 180,E1 -1139.672,E2 -1139.672} C_VEL
LIN {X 0,Y 594.374,Z 510.452,A -85,B 0,C 180,E1 -1142.54,E2 -1142.54} C_VEL
LIN {X 0,Y 594.375,Z 510.448,A -85,B 0,C 180,E1 -1144.808,E2 -1144.808} C_VEL
LIN {X 0,Y 594.392,Z 510.529,A -85,B 0,C 180,E1 -1147.411,E2 -1147.411} C_VEL
LIN {X 0,Y 594.722,Z 515.506,A -85,B 0,C 180,E1 -1148.146,E2 -1148.146} C_VEL
LIN {X 0,Y 594.592,Z 535.52,A -85,B 0,C 180,E1 -1151.013,E2 -1151.013} C_VEL
LIN {X 0,Y 594.505,Z 554.544,A -85,B 0,C 180,E1 -1153.695,E2 -1153.695} C_VEL
LIN {X 0,Y 594.433,Z 574.693,A -85,B 0,C 180,E1 -1156.497,E2 -1156.497} C_VEL
LIN {X 0,Y 594.469,Z 576.169,A -85,B 0,C 180,E1 -1156.672,E2 -1156.672} C_VEL
LIN {X 0,Y 594.769,Z 581.535,A -85,B 0,C 180,E1 -1156.744,E2 -1156.744} C_VEL
LIN {X 0,Y 594.654,Z 683.962,A -85,B 0,C 180,E1 -1157.999,E2 -1157.999} C_VEL
LIN {X 0,Y 594.621,Z 697.228,A -85,B 0,C 180,E1 -1158.301,E2 -1158.301} C_VEL
LIN {X 0,Y 594.577,Z 709.579,A -85,B 0,C 180,E1 -1158.719,E2 -1158.719} C_VEL
LIN {X 0,Y 594.538,Z 721.638,A -85,B 0,C 180,E1 -1159.27,E2 -1159.27} C_VEL
LIN {X 0,Y 594.468,Z 733.203,A -85,B 0,C 180,E1 -1159.958,E2 -1159.958} C_VEL
LIN {X 0,Y 594.413,Z 743.599,A -85,B 0,C 180,E1 -1160.73,E2 -1160.73} C_VEL
LIN {X 0,Y 594.383,Z 752.114,A -85,B 0,C 180,E1 -1161.501,E2 -1161.501} C_VEL
LIN {X 0,Y 594.347,Z 759.962,A -85,B 0,C 180,E1 -1162.356,E2 -1162.356} C_VEL
LIN {X 0,Y 594.282,Z 767.813,A -85,B 0,C 180,E1 -1163.408,E2 -1163.408} C_VEL
LIN {X 0,Y 594.289,Z 774.681,A -85,B 0,C 180,E1 -1164.571,E2 -1164.571} C_VEL
LIN {X 0,Y 594.27,Z 779.372,A -85,B 0,C 180,E1 -1165.591,E2 -1165.591} C_VEL
LIN {X 0,Y 594.268,Z 782.956,A -85,B 0,C 180,E1 -1166.61,E2 -1166.61} C_VEL
LIN {X 0,Y 594.226,Z 784.809,A -85,B 0,C 180,E1 -1167.288,E2 -1167.288} C_VEL
LIN {X 0,Y 594.239,Z 786.202,A -85,B 0,C 180,E1 -1167.967,E2 -1167.967} C_VEL
LIN {X 0,Y 594.239,Z 787.784,A -85,B 0,C 180,E1 -1169.322,E2 -1169.322} C_VEL
LIN {X 0,Y 594.236,Z 788,A -85,B 0,C 180,E1 -1170,E2 -1170} C_VEL
LIN {X 0,Y 594.247,Z 787.185,A -85,B 0,C 180,E1 -1171.355,E2 -1171.355} C_VEL
LIN {X 0,Y 594.239,Z 786.202,A -85,B 0,C 180,E1 -1172.033,E2 -1172.033} C_VEL
LIN {X 0,Y 594.226,Z 784.81,A -85,B 0,C 180,E1 -1172.712,E2 -1172.712} C_VEL
LIN {X 0,Y 594.288,Z 781.896,A -85,B 0,C 180,E1 -1173.729,E2 -1173.729} C_VEL
LIN {X 0,Y 594.242,Z 777.95,A -85,B 0,C 180,E1 -1174.749,E2 -1174.749} C_VEL
LIN {X 0,Y 594.304,Z 771.878,A -85,B 0,C 180,E1 -1175.939,E2 -1175.939} C_VEL
LIN {X 0,Y 594.308,Z 765.237,A -85,B 0,C 180,E1 -1176.962,E2 -1176.962} C_VEL
LIN {X 0,Y 594.359,Z 756.991,A -85,B 0,C 180,E1 -1177.986,E2 -1177.986} C_VEL
LIN {X 0,Y 594.382,Z 748.539,A -85,B 0,C 180,E1 -1178.842,E2 -1178.842} C_VEL
LIN {X 0,Y 594.423,Z 738.096,A -85,B 0,C 180,E1 -1179.699,E2 -1179.699} C_VEL
LIN {X 0,Y 594.485,Z 727.763,A -85,B 0,C 180,E1 -1180.386,E2 -1180.386} C_VEL
LIN {X 0,Y 594.56,Z 716.696,A -85,B 0,C 180,E1 -1180.974,E2 -1180.974} C_VEL
LIN {X 0,Y 594.594,Z 704.709,A -85,B 0,C 180,E1 -1181.464,E2 -1181.464} C_VEL
LIN {X 0,Y 594.635,Z 691.363,A -85,B 0,C 180,E1 -1181.85,E2 -1181.85} C_VEL
LIN {X 0,Y 594.691,Z 678.106,A -85,B 0,C 180,E1 -1182.087,E2 -1182.087} C_VEL
LIN {X 0,Y 594.631,Z 577.288,A -85,B 0,C 180,E1 -1183.311,E2 -1183.311} C_VEL
LIN {X 0,Y 594.45,Z 575.795,A -85,B 0,C 180,E1 -1183.35,E2 -1183.35} C_VEL
LIN {X 0,Y 594.506,Z 554.544,A -85,B 0,C 180,E1 -1186.305,E2 -1186.305} C_VEL
LIN {X 0,Y 594.631,Z 534.726,A -85,B 0,C 180,E1 -1189.099,E2 -1189.099} C_VEL
LIN {X 0,Y 594.742,Z 514.246,A -85,B 0,C 180,E1 -1192.035,E2 -1192.035} C_VEL
LIN {X 0,Y 594.389,Z 510.445,A -85,B 0,C 180,E1 -1192.624,E2 -1192.624} C_VEL
LIN {X 0,Y 594.375,Z 510.448,A -85,B 0,C 180,E1 -1195.192,E2 -1195.192} C_VEL
LIN {X 0,Y 594.386,Z 510.45,A -85,B 0,C 180,E1 -1197.526,E2 -1197.526} C_VEL
LIN {X 0,Y 594.387,Z 510.44,A -85,B 0,C 180,E1 -1200.328,E2 -1200.328} C_VEL
LIN {X 0,Y 594.378,Z 510.443,A -85,B 0,C 180,E1 -1202.949,E2 -1202.949} C_VEL
LIN {X 0,Y 594.349,Z 510.454,A -85,B 0,C 180,E1 -1205.408,E2 -1205.408} C_VEL
LIN {X 0,Y 594.386,Z 510.442,A -85,B 0,C 180,E1 -1207.94,E2 -1207.94} C_VEL
LIN {X 0,Y 594.378,Z 510.442,A -85,B 0,C 180,E1 -1210.822,E2 -1210.822} C_VEL
LIN {X 0,Y 594.378,Z 510.445,A -85,B 0,C 180,E1 -1213.84,E2 -1213.84} C_VEL
LIN {X 0,Y 594.361,Z 510.443,A -85,B 0,C 180,E1 -1216.7,E2 -1216.7} C_VEL
LIN {X 0,Y 594.368,Z 510.452,A -85,B 0,C 180,E1 -1219.433,E2 -1219.433} C_VEL
LIN {X 0,Y 594.383,Z 510.44,A -85,B 0,C 180,E1 -1222.391,E2 -1222.391} C_VEL
LIN {X 0,Y 594.381,Z 510.44,A -85,B 0,C 180,E1 -1224.67,E2 -1224.67} C_VEL
LIN {X 0,Y 594.372,Z 510.445,A -85,B 0,C 180,E1 -1227.087,E2 -1227.087} C_VEL
LIN {X 0,Y 594.393,Z 510.445,A -85,B 0,C 180,E1 -1229.669,E2 -1229.669} C_VEL
LIN {X 0,Y 594.365,Z 510.442,A -85,B 0,C 180,E1 -1232.539,E2 -1232.539} C_VEL
LIN {X 0,Y 594.374,Z 510.442,A -85,B 0,C 180,E1 -1234.807,E2 -1234.807} C_VEL
LIN {X 0,Y 594.356,Z 510.45,A -85,B 0,C 180,E1 -1237.264,E2 -1237.264} C_VEL
LIN {X 0,Y 594.37,Z 510.444,A -85,B 0,C 180,E1 -1239.946,E2 -1239.946} C_VEL
LIN {X 0,Y 594.383,Z 510.441,A -85,B 0,C 180,E1 -1242.806,E2 -1242.806} C_VEL
LIN {X 0,Y 594.378,Z 510.445,A -85,B 0,C 180,E1 -1245.826,E2 -1245.826} C_VEL
LIN {X 0,Y 594.385,Z 510.439,A -85,B 0,C 180,E1 -1248.404,E2 -1248.404} C_VEL
LIN {X 0,Y 594.394,Z 510.444,A -85,B 0,C 180,E1 -1251.158,E2 -1251.158} C_VEL
LIN {X 0,Y 594.362,Z 510.446,A -85,B 0,C 180,E1 -1253.891,E2 -1253.891} C_VEL
LIN {X 0,Y 594.378,Z 510.441,A -85,B 0,C 180,E1 -1256.611,E2 -1256.611} C_VEL
LIN {X 0,Y 594.416,Z 510.444,A -85,B 0,C 180,E1 -1259.323,E2 -1259.323} C_VEL
LIN {X 0,Y 594.388,Z 510.441,A -85,B 0,C 180,E1 -1262.033,E2 -1262.033} C_VEL
LIN {X 0,Y 594.397,Z 510.439,A -85,B 0,C 180,E1 -1264.748,E2 -1264.748} C_VEL
LIN {X 0,Y 594.394,Z 510.449,A -85,B 0,C 180,E1 -1267.473,E2 -1267.473} C_VEL
LIN {X 0,Y 594.387,Z 510.44,A -85,B 0,C 180,E1 -1270.216,E2 -1270.216} C_VEL
LIN {X 0,Y 594.365,Z 510.445,A -85,B 0,C 180,E1 -1272.983,E2 -1272.983} C_VEL
LIN {X 0,Y 594.357,Z 510.446,A -85,B 0,C 180,E1 -1275.339,E2 -1275.339} C_VEL
LIN {X 0,Y 593.686,Z 510.531,A -85,B 0,C 180,E1 -1275.905,E2 -1275.905} C_VEL
LIN {X 0,Y 590.831,Z 510.885,A -85,B 0,C 180,E1 -1276.823,E2 -1276.823} C_VEL
LIN {X 0,Y 588.426,Z 511.19,A -85,B 0,C 180,E1 -1277.562,E2 -1277.562} C_VEL
LIN {X 0,Y 587.399,Z 511.311,A -85,B 0,C 180,E1 -1278.132,E2 -1278.132} C_VEL
LIN {X 0,Y 587.319,Z 511.32,A -85,B 0,C 180,E1 -1278.325,E2 -1278.325} C_VEL
LIN {X 0,Y 587.349,Z 511.32,A -85,B 0,C 180,E1 -1281.045,E2 -1281.045} C_VEL
LIN {X 0,Y 587.33,Z 511.32,A -85,B 0,C 180,E1 -1284.007,E2 -1284.007} C_VEL
LIN {X 0,Y 587.357,Z 511.315,A -85,B 0,C 180,E1 -1286.278,E2 -1286.278} C_VEL
LIN {X 0,Y 587.347,Z 511.322,A -85,B 0,C 180,E1 -1289.135,E2 -1289.135} C_VEL
LIN {X 0,Y 587.35,Z 511.32,A -85,B 0,C 180,E1 -1291.839,E2 -1291.839} C_VEL
LIN {X 0,Y 587.353,Z 511.315,A -85,B 0,C 180,E1 -1294.35,E2 -1294.35} C_VEL
LIN {X 0,Y 587.347,Z 511.317,A -85,B 0,C 180,E1 -1296.747,E2 -1296.747} C_VEL
LIN {X 0,Y 587.342,Z 511.327,A -85,B 0,C 180,E1 -1299.36,E2 -1299.36} C_VEL
LIN {X 0,Y 587.33,Z 511.319,A -85,B 0,C 180,E1 -1302.109,E2 -1302.109} C_VEL
LIN {X 0,Y 587.312,Z 511.326,A -85,B 0,C 180,E1 -1305.09,E2 -1305.09} C_VEL
LIN {X 0,Y 587.35,Z 511.318,A -85,B 0,C 180,E1 -1307.929,E2 -1307.929} C_VEL
LIN {X 0,Y 587.332,Z 511.323,A -85,B 0,C 180,E1 -1311.059,E2 -1311.059} C_VEL
LIN {X 0,Y 587.352,Z 511.325,A -85,B 0,C 180,E1 -1313.293,E2 -1313.293} C_VEL
LIN {X 0,Y 587.361,Z 511.319,A -85,B 0,C 180,E1 -1315.781,E2 -1315.781} C_VEL
LIN {X 0,Y 587.348,Z 511.316,A -85,B 0,C 180,E1 -1318.232,E2 -1318.232} C_VEL
LIN {X 0,Y 587.35,Z 511.318,A -85,B 0,C 180,E1 -1320.867,E2 -1320.867} C_VEL
LIN {X 0,Y 587.359,Z 511.318,A -85,B 0,C 180,E1 -1323.82,E2 -1323.82} C_VEL
LIN {X 0,Y 587.332,Z 511.32,A -85,B 0,C 180,E1 -1325.994,E2 -1325.994} C_VEL
LIN {X 0,Y 587.324,Z 511.32,A -85,B 0,C 180,E1 -1328.226,E2 -1328.226} C_VEL
LIN {X 0,Y 587.354,Z 511.323,A -85,B 0,C 180,E1 -1331.152,E2 -1331.152} C_VEL
LIN {X 0,Y 587.329,Z 511.323,A -85,B 0,C 180,E1 -1334.025,E2 -1334.025} C_VEL
LIN {X 0,Y 587.382,Z 511.474,A -85,B 0,C 180,E1 -1334.472,E2 -1334.472} C_VEL
LIN {X 0,Y 587.502,Z 521.22,A -85,B 0,C 180,E1 -1336.158,E2 -1336.158} C_VEL
LIN {X 0,Y 587.414,Z 538.728,A -85,B 0,C 180,E1 -1339.139,E2 -1339.139} C_VEL
LIN {X 0,Y 587.344,Z 547.121,A -85,B 0,C 180,E1 -1340.552,E2 -1340.552} C_VEL
LIN {X 0,Y 587.87,Z 551.157,A -85,B 0,C 180,E1 -1340.626,E2 -1340.626} C_VEL
LIN {X 0,Y 587.722,Z 654.019,A -85,B 0,C 180,E1 -1341.901,E2 -1341.901} C_VEL
LIN {X 0,Y 587.678,Z 667.142,A -85,B 0,C 180,E1 -1342.203,E2 -1342.203} C_VEL
LIN {X 0,Y 587.603,Z 679.637,A -85,B 0,C 180,E1 -1342.63,E2 -1342.63} C_VEL
LIN {X 0,Y 587.566,Z 690.558,A -85,B 0,C 180,E1 -1343.13,E2 -1343.13} C_VEL
LIN {X 0,Y 587.469,Z 702.282,A -85,B 0,C 180,E1 -1343.819,E2 -1343.819} C_VEL
LIN {X 0,Y 587.377,Z 712.754,A -85,B 0,C 180,E1 -1344.593,E2 -1344.593} C_VEL
LIN {X 0,Y 587.327,Z 723.066,A -85,B 0,C 180,E1 -1345.539,E2 -1345.539} C_VEL
LIN {X 0,Y 587.231,Z 732.034,A -85,B 0,C 180,E1 -1346.569,E2 -1346.569} C_VEL
LIN {X 0,Y 587.262,Z 739.274,A -85,B 0,C 180,E1 -1347.599,E2 -1347.599} C_VEL
LIN {X 0,Y 587.171,Z 745.09,A -85,B 0,C 180,E1 -1348.628,E2 -1348.628} C_VEL
LIN {X 0,Y 587.205,Z 749.677,A -85,B 0,C 180,E1 -1349.657,E2 -1349.657} C_VEL
LIN {X 0,Y 587.143,Z 753.179,A -85,B 0,C 180,E1 -1350.686,E2 -1350.686} C_VEL
LIN {X 0,Y 587.148,Z 754.97,A -85,B 0,C 180,E1 -1351.372,E2 -1351.372} C_VEL
LIN {X 0,Y 587.14,Z 756.316,A -85,B 0,C 180,E1 -1352.058,E2 -1352.058} C_VEL
LIN {X 0,Y 587.181,Z 757.833,A -85,B 0,C 180,E1 -1353.431,E2 -1353.431} C_VEL
LIN {X 0,Y 587.17,Z 757.99,A -85,B 0,C 180,E1 -1354.118,E2 -1354.118} C_VEL
LIN {X 0,Y 587.17,Z 757.096,A -85,B 0,C 180,E1 -1355.495,E2 -1355.495} C_VEL
LIN {X 0,Y 587.188,Z 755.274,A -85,B 0,C 180,E1 -1356.574,E2 -1356.574} C_VEL
LIN {X 0,Y 587.173,Z 751.582,A -85,B 0,C 180,E1 -1357.911,E2 -1357.911} C_VEL
LIN {X 0,Y 587.159,Z 747.508,A -85,B 0,C 180,E1 -1358.952,E2 -1358.952} C_VEL
LIN {X 0,Y 587.215,Z 741.224,A -85,B 0,C 180,E1 -1360.168,E2 -1360.168} C_VEL
LIN {X 0,Y 587.264,Z 734.486,A -85,B 0,C 180,E1 -1361.196,E2 -1361.196} C_VEL
LIN {X 0,Y 587.312,Z 727.336,A -85,B 0,C 180,E1 -1362.088,E2 -1362.088} C_VEL
LIN {X 0,Y 587.344,Z 718.852,A -85,B 0,C 180,E1 -1362.965,E2 -1362.965} C_VEL
LIN {X 0,Y 587.422,Z 708.327,A -85,B 0,C 180,E1 -1363.844,E2 -1363.844} C_VEL
LIN {X 0,Y 587.491,Z 697.876,A -85,B 0,C 180,E1 -1364.549,E2 -1364.549} C_VEL
LIN {X 0,Y 587.588,Z 686.373,A -85,B 0,C 180,E1 -1365.167,E2 -1365.167} C_VEL
LIN {X 0,Y 587.657,Z 674.483,A -85,B 0,C 180,E1 -1365.654,E2 -1365.654} C_VEL
LIN {X 0,Y 587.701,Z 661.608,A -85,B 0,C 180,E1 -1366.031,E2 -1366.031} C_VEL
LIN {X 0,Y 587.758,Z 648.244,A -85,B 0,C 180,E1 -1366.275,E2 -1366.275} C_VEL
LIN {X 0,Y 587.799,Z 549.888,A -85,B 0,C 180,E1 -1367.482,E2 -1367.482} C_VEL
LIN {X 0,Y 587.357,Z 547.106,A -85,B 0,C 180,E1 -1367.54,E2 -1367.54} C_VEL
LIN {X 0,Y 587.449,Z 530.774,A -85,B 0,C 180,E1 -1370.3,E2 -1370.3} C_VEL
LIN {X 0,Y 587.558,Z 513.573,A -85,B 0,C 180,E1 -1373.248,E2 -1373.248} C_VEL
LIN {X 0,Y 587.368,Z 511.319,A -85,B 0,C 180,E1 -1373.677,E2 -1373.677} C_VEL
LIN {X 0,Y 587.34,Z 511.322,A -85,B 0,C 180,E1 -1376.278,E2 -1376.278} C_VEL
LIN {X 0,Y 587.351,Z 511.32,A -85,B 0,C 180,E1 -1379.133,E2 -1379.133} C_VEL
LIN {X 0,Y 587.351,Z 511.316,A -85,B 0,C 180,E1 -1381.836,E2 -1381.836} C_VEL
LIN {X 0,Y 587.35,Z 511.321,A -85,B 0,C 180,E1 -1384.347,E2 -1384.347} C_VEL
LIN {X 0,Y 587.353,Z 511.325,A -85,B 0,C 180,E1 -1386.746,E2 -1386.746} C_VEL
LIN {X 0,Y 587.344,Z 511.318,A -85,B 0,C 180,E1 -1389.358,E2 -1389.358} C_VEL
LIN {X 0,Y 587.334,Z 511.32,A -85,B 0,C 180,E1 -1392.107,E2 -1392.107} C_VEL
LIN {X 0,Y 587.312,Z 511.324,A -85,B 0,C 180,E1 -1395.088,E2 -1395.088} C_VEL
LIN {X 0,Y 587.348,Z 511.317,A -85,B 0,C 180,E1 -1397.927,E2 -1397.927} C_VEL
LIN {X 0,Y 587.33,Z 511.323,A -85,B 0,C 180,E1 -1401.057,E2 -1401.057} C_VEL
LIN {X 0,Y 587.348,Z 511.318,A -85,B 0,C 180,E1 -1403.291,E2 -1403.291} C_VEL
LIN {X 0,Y 587.365,Z 511.314,A -85,B 0,C 180,E1 -1405.78,E2 -1405.78} C_VEL
LIN {X 0,Y 587.347,Z 511.32,A -85,B 0,C 180,E1 -1408.231,E2 -1408.231} C_VEL
LIN {X 0,Y 587.347,Z 511.323,A -85,B 0,C 180,E1 -1410.865,E2 -1410.865} C_VEL
LIN {X 0,Y 587.356,Z 511.315,A -85,B 0,C 180,E1 -1413.817,E2 -1413.817} C_VEL
LIN {X 0,Y 587.316,Z 511.329,A -85,B 0,C 180,E1 -1416.741,E2 -1416.741} C_VEL
LIN {X 0,Y 587.326,Z 511.319,A -85,B 0,C 180,E1 -1419.695,E2 -1419.695} C_VEL
LIN {X 0,Y 587.352,Z 511.325,A -85,B 0,C 180,E1 -1422.594,E2 -1422.594} C_VEL
LIN {X 0,Y 587.354,Z 511.315,A -85,B 0,C 180,E1 -1425.739,E2 -1425.739} C_VEL
LIN {X 0,Y 587.352,Z 511.322,A -85,B 0,C 180,E1 -1428.858,E2 -1428.858} C_VEL
LIN {X 0,Y 587.363,Z 511.314,A -85,B 0,C 180,E1 -1431.745,E2 -1431.745} C_VEL
LIN {X 0,Y 587.352,Z 511.324,A -85,B 0,C 180,E1 -1434.507,E2 -1434.507} C_VEL
LIN {X 0,Y 587.374,Z 511.314,A -85,B 0,C 180,E1 -1437.257,E2 -1437.257} C_VEL
LIN {X 0,Y 587.373,Z 511.315,A -85,B 0,C 180,E1 -1440,E2 -1440} C_VEL
LIN {X 0,Y 587.376,Z 511.32,A -85,B 0,C 180,E1 -1442.743,E2 -1442.743} C_VEL
LIN {X 0,Y 587.351,Z 511.316,A -85,B 0,C 180,E1 -1445.493,E2 -1445.493} C_VEL
LIN {X 0,Y 587.364,Z 511.319,A -85,B 0,C 180,E1 -1448.255,E2 -1448.255} C_VEL
LIN {X 0,Y 587.352,Z 511.318,A -85,B 0,C 180,E1 -1451.142,E2 -1451.142} C_VEL
LIN {X 0,Y 587.354,Z 511.32,A -85,B 0,C 180,E1 -1454.261,E2 -1454.261} C_VEL
LIN {X 0,Y 587.35,Z 511.316,A -85,B 0,C 180,E1 -1457.406,E2 -1457.406} C_VEL
LIN {X 0,Y 587.325,Z 511.325,A -85,B 0,C 180,E1 -1460.305,E2 -1460.305} C_VEL
LIN {X 0,Y 587.315,Z 511.321,A -85,B 0,C 180,E1 -1463.259,E2 -1463.259} C_VEL
LIN {X 0,Y 587.333,Z 511.318,A -85,B 0,C 180,E1 -1465.517,E2 -1465.517} C_VEL
LIN {X 0,Y 587.341,Z 511.317,A -85,B 0,C 180,E1 -1467.818,E2 -1467.818} C_VEL
LIN {X 0,Y 587.342,Z 511.327,A -85,B 0,C 180,E1 -1470.513,E2 -1470.513} C_VEL
LIN {X 0,Y 587.329,Z 511.319,A -85,B 0,C 180,E1 -1473.397,E2 -1473.397} C_VEL
LIN {X 0,Y 587.351,Z 511.317,A -85,B 0,C 180,E1 -1475.896,E2 -1475.896} C_VEL
LIN {X 0,Y 587.327,Z 511.328,A -85,B 0,C 180,E1 -1478.48,E2 -1478.48} C_VEL
LIN {X 0,Y 587.331,Z 511.32,A -85,B 0,C 180,E1 -1481.158,E2 -1481.158} C_VEL
LIN {X 0,Y 587.321,Z 511.323,A -85,B 0,C 180,E1 -1484.114,E2 -1484.114} C_VEL
LIN {X 0,Y 587.319,Z 511.323,A -85,B 0,C 180,E1 -1486.995,E2 -1486.995} C_VEL
LIN {X 0,Y 587.317,Z 511.321,A -85,B 0,C 180,E1 -1489.747,E2 -1489.747} C_VEL
LIN {X 0,Y 587.345,Z 511.325,A -85,B 0,C 180,E1 -1492.393,E2 -1492.393} C_VEL
LIN {X 0,Y 587.346,Z 511.317,A -85,B 0,C 180,E1 -1495.653,E2 -1495.653} C_VEL
LIN {X 0,Y 587.352,Z 511.322,A -85,B 0,C 180,E1 -1498.233,E2 -1498.233} C_VEL
LIN {X 0,Y 587.349,Z 511.321,A -85,B 0,C 180,E1 -1500.867,E2 -1500.867} C_VEL
LIN {X 0,Y 587.358,Z 511.317,A -85,B 0,C 180,E1 -1503.82,E2 -1503.82} C_VEL
LIN {X 0,Y 587.338,Z 511.322,A -85,B 0,C 180,E1 -1505.994,E2 -1505.994} C_VEL
LIN {X 0,Y 587.344,Z 511.446,A -85,B 0,C 180,E1 -1507.26,E2 -1507.26} C_VEL
LIN {X 0,Y 587.822,Z 515.506,A -85,B 0,C 180,E1 -1507.876,E2 -1507.876} C_VEL
LIN {X 0,Y 587.67,Z 536.133,A -85,B 0,C 180,E1 -1510.869,E2 -1510.869} C_VEL
LIN {X 0,Y 587.511,Z 555.803,A -85,B 0,C 180,E1 -1513.674,E2 -1513.674} C_VEL
LIN {X 0,Y 587.389,Z 575.795,A -85,B 0,C 180,E1 -1516.486,E2 -1516.486} C_VEL
LIN {X 0,Y 587.886,Z 579.746,A -85,B 0,C 180,E1 -1516.564,E2 -1516.564} C_VEL
LIN {X 0,Y 587.716,Z 683.962,A -85,B 0,C 180,E1 -1517.855,E2 -1517.855} C_VEL
LIN {X 0,Y 587.666,Z 697.228,A -85,B 0,C 180,E1 -1518.161,E2 -1518.161} C_VEL
LIN {X 0,Y 587.605,Z 709.758,A -85,B 0,C 180,E1 -1518.59,E2 -1518.59} C_VEL
LIN {X 0,Y 587.554,Z 721.636,A -85,B 0,C 180,E1 -1519.141,E2 -1519.141} C_VEL
LIN {X 0,Y 587.458,Z 733.204,A -85,B 0,C 180,E1 -1519.837,E2 -1519.837} C_VEL
LIN {X 0,Y 587.391,Z 743.6,A -85,B 0,C 180,E1 -1520.618,E2 -1520.618} C_VEL
LIN {X 0,Y 587.321,Z 752.114,A -85,B 0,C 180,E1 -1521.398,E2 -1521.398} C_VEL
LIN {X 0,Y 587.273,Z 759.962,A -85,B 0,C 180,E1 -1522.263,E2 -1522.263} C_VEL
LIN {X 0,Y 587.23,Z 766.471,A -85,B 0,C 180,E1 -1523.127,E2 -1523.127} C_VEL
LIN {X 0,Y 587.236,Z 772.867,A -85,B 0,C 180,E1 -1524.161,E2 -1524.161} C_VEL
LIN {X 0,Y 587.147,Z 777.95,A -85,B 0,C 180,E1 -1525.194,E2 -1525.194} C_VEL
LIN {X 0,Y 587.212,Z 781.896,A -85,B 0,C 180,E1 -1526.226,E2 -1526.226} C_VEL
LIN {X 0,Y 587.132,Z 784.809,A -85,B 0,C 180,E1 -1527.256,E2 -1527.256} C_VEL
LIN {X 0,Y 587.138,Z 786.201,A -85,B 0,C 180,E1 -1527.942,E2 -1527.942} C_VEL
LIN {X 0,Y 587.14,Z 787.784,A -85,B 0,C 180,E1 -1529.314,E2 -1529.314} C_VEL
LIN {X 0,Y 587.137,Z 788,A -85,B 0,C 180,E1 -1530,E2 -1530} C_VEL
LIN {X 0,Y 587.147,Z 787.185,A -85,B 0,C 180,E1 -1531.372,E2 -1531.372} C_VEL
LIN {X 0,Y 587.138,Z 786.201,A -85,B 0,C 180,E1 -1532.058,E2 -1532.058} C_VEL
LIN {X 0,Y 587.132,Z 784.81,A -85,B 0,C 180,E1 -1532.744,E2 -1532.744} C_VEL
LIN {X 0,Y 587.212,Z 781.896,A -85,B 0,C 180,E1 -1533.774,E2 -1533.774} C_VEL
LIN {X 0,Y 587.147,Z 777.95,A -85,B 0,C 180,E1 -1534.806,E2 -1534.806} C_VEL
LIN {X 0,Y 587.217,Z 771.878,A -85,B 0,C 180,E1 -1536.011,E2 -1536.011} C_VEL
LIN {X 0,Y 587.245,Z 765.238,A -85,B 0,C 180,E1 -1537.046,E2 -1537.046} C_VEL
LIN {X 0,Y 587.299,Z 756.992,A -85,B 0,C 180,E1 -1538.083,E2 -1538.083} C_VEL
LIN {X 0,Y 587.343,Z 748.54,A -85,B 0,C 180,E1 -1538.949,E2 -1538.949} C_VEL
LIN {X 0,Y 587.41,Z 738.098,A -85,B 0,C 180,E1 -1539.816,E2 -1539.816} C_VEL
LIN {X 0,Y 587.505,Z 727.763,A -85,B 0,C 180,E1 -1540.511,E2 -1540.511} C_VEL
LIN {X 0,Y 587.583,Z 715.806,A -85,B 0,C 180,E1 -1541.149,E2 -1541.149} C_VEL
LIN {X 0,Y 587.624,Z 703.598,A -85,B 0,C 180,E1 -1541.639,E2 -1541.639} C_VEL
LIN {X 0,Y 587.683,Z 690.448,A -85,B 0,C 180,E1 -1542.014,E2 -1542.014} C_VEL
LIN {X 0,Y 587.772,Z 678.106,A -85,B 0,C 180,E1 -1542.231,E2 -1542.231} C_VEL
LIN {X 0,Y 587.712,Z 577.856,A -85,B 0,C 180,E1 -1543.464,E2 -1543.464} C_VEL
LIN {X 0,Y 587.389,Z 575.795,A -85,B 0,C 180,E1 -1543.514,E2 -1543.514} C_VEL
LIN {X 0,Y 587.529,Z 555.803,A -85,B 0,C 180,E1 -1546.326,E2 -1546.326} C_VEL
LIN {X 0,Y 587.67,Z 536.133,A -85,B 0,C 180,E1 -1549.131,E2 -1549.131} C_VEL
LIN {X 0,Y 587.822,Z 515.506,A -85,B 0,C 180,E1 -1552.124,E2 -1552.124} C_VEL
LIN {X 0,Y 587.331,Z 511.326,A -85,B 0,C 180,E1 -1552.791,E2 -1552.791} C_VEL
LIN {X 0,Y 587.332,Z 511.329,A -85,B 0,C 180,E1 -1555.516,E2 -1555.516} C_VEL
LIN {X 0,Y 587.348,Z 511.321,A -85,B 0,C 180,E1 -1557.817,E2 -1557.817} C_VEL
LIN {X 0,Y 587.342,Z 511.317,A -85,B 0,C 180,E1 -1560.51,E2 -1560.51} C_VEL
LIN {X 0,Y 587.339,Z 511.322,A -85,B 0,C 180,E1 -1563.111,E2 -1563.111} C_VEL
LIN {X 0,Y 587.323,Z 511.329,A -85,B 0,C 180,E1 -1565.541,E2 -1565.541} C_VEL
LIN {X 0,Y 587.34,Z 511.321,A -85,B 0,C 180,E1 -1567.838,E2 -1567.838} C_VEL
LIN {X 0,Y 587.317,Z 511.32,A -85,B 0,C 180,E1 -1570.253,E2 -1570.253} C_VEL
LIN {X 0,Y 587.322,Z 511.324,A -85,B 0,C 180,E1 -1573.119,E2 -1573.119} C_VEL
LIN {X 0,Y 587.317,Z 511.322,A -85,B 0,C 180,E1 -1576.049,E2 -1576.049} C_VEL
LIN {X 0,Y 587.331,Z 511.321,A -85,B 0,C 180,E1 -1578.924,E2 -1578.924} C_VEL
LIN {X 0,Y 587.327,Z 511.329,A -85,B 0,C 180,E1 -1581.52,E2 -1581.52} C_VEL
LIN {X 0,Y 587.347,Z 511.316,A -85,B 0,C 180,E1 -1584.454,E2 -1584.454} C_VEL
LIN {X 0,Y 587.333,Z 511.32,A -85,B 0,C 180,E1 -1586.887,E2 -1586.887} C_VEL
LIN {X 0,Y 587.343,Z 511.327,A -85,B 0,C 180,E1 -1589.487,E2 -1589.487} C_VEL
LIN {X 0,Y 587.343,Z 511.317,A -85,B 0,C 180,E1 -1592.306,E2 -1592.306} C_VEL
LIN {X 0,Y 587.334,Z 511.318,A -85,B 0,C 180,E1 -1594.483,E2 -1594.483} C_VEL
LIN {X 0,Y 587.332,Z 511.328,A -85,B 0,C 180,E1 -1597.486,E2 -1597.486} C_VEL
LIN {X 0,Y 587.325,Z 511.325,A -85,B 0,C 180,E1 -1599.695,E2 -1599.695} C_VEL
LIN {X 0,Y 587.35,Z 511.316,A -85,B 0,C 180,E1 -1602.594,E2 -1602.594} C_VEL
LIN {X 0,Y 587.354,Z 511.321,A -85,B 0,C 180,E1 -1605.739,E2 -1605.739} C_VEL
LIN {X 0,Y 587.352,Z 511.318,A -85,B 0,C 180,E1 -1608.858,E2 -1608.858} C_VEL
LIN {X 0,Y 587.363,Z 511.32,A -85,B 0,C 180,E1 -1611.745,E2 -1611.745} C_VEL
LIN {X 0,Y 587.351,Z 511.316,A -85,B 0,C 180,E1 -1614.507,E2 -1614.507} C_VEL
LIN {X 0,Y 587.376,Z 511.32,A -85,B 0,C 180,E1 -1617.257,E2 -1617.257} C_VEL
LIN {X 0,Y 587.373,Z 511.315,A -85,B 0,C 180,E1 -1620,E2 -1620} C_VEL
LIN {X 0,Y 587.374,Z 511.314,A -85,B 0,C 180,E1 -1622.743,E2 -1622.743} C_VEL
LIN {X 0,Y 587.351,Z 511.326,A -85,B 0,C 180,E1 -1625.493,E2 -1625.493} C_VEL
LIN {X 0,Y 587.364,Z 511.314,A -85,B 0,C 180,E1 -1628.255,E2 -1628.255} C_VEL
LIN {X 0,Y 587.352,Z 511.321,A -85,B 0,C 180,E1 -1631.142,E2 -1631.142} C_VEL
LIN {X 0,Y 587.354,Z 511.316,A -85,B 0,C 180,E1 -1634.261,E2 -1634.261} C_VEL
LIN {X 0,Y 587.35,Z 511.327,A -85,B 0,C 180,E1 -1637.406,E2 -1637.406} C_VEL
LIN {X 0,Y 587.319,Z 511.32,A -85,B 0,C 180,E1 -1638.325,E2 -1638.325} C_VEL
LIN {X 0,Y 586.667,Z 511.404,A -85,B 0,C 180,E1 -1638.897,E2 -1638.897} C_VEL
LIN {X 0,Y 583.837,Z 511.764,A -85,B 0,C 180,E1 -1639.825,E2 -1639.825} C_VEL
LIN {X 0,Y 581.428,Z 512.068,A -85,B 0,C 180,E1 -1640.572,E2 -1640.572} C_VEL
LIN {X 0,Y 580.375,Z 512.195,A -85,B 0,C 180,E1 -1641.149,E2 -1641.149} C_VEL
LIN {X 0,Y 580.28,Z 512.205,A -85,B 0,C 180,E1 -1641.344,E2 -1641.344} C_VEL
LIN {X 0,Y 580.293,Z 512.195,A -85,B 0,C 180,E1 -1644.317,E2 -1644.317} C_VEL
LIN {X 0,Y 580.303,Z 512.194,A -85,B 0,C 180,E1 -1646.622,E2 -1646.622} C_VEL
LIN {X 0,Y 580.301,Z 512.203,A -85,B 0,C 180,E1 -1649.312,E2 -1649.312} C_VEL
LIN {X 0,Y 580.297,Z 512.195,A -85,B 0,C 180,E1 -1652.201,E2 -1652.201} C_VEL
LIN {X 0,Y 580.298,Z 512.195,A -85,B 0,C 180,E1 -1654.696,E2 -1654.696} C_VEL
LIN {X 0,Y 580.295,Z 512.203,A -85,B 0,C 180,E1 -1657.269,E2 -1657.269} C_VEL
LIN {X 0,Y 580.294,Z 512.195,A -85,B 0,C 180,E1 -1660.272,E2 -1660.272} C_VEL
LIN {X 0,Y 580.273,Z 512.198,A -85,B 0,C 180,E1 -1662.707,E2 -1662.707} C_VEL
LIN {X 0,Y 580.271,Z 512.205,A -85,B 0,C 180,E1 -1665.609,E2 -1665.609} C_VEL
LIN {X 0,Y 580.312,Z 512.193,A -85,B 0,C 180,E1 -1668.235,E2 -1668.235} C_VEL
LIN {X 0,Y 580.287,Z 512.199,A -85,B 0,C 180,E1 -1670.967,E2 -1670.967} C_VEL
LIN {X 0,Y 580.277,Z 512.204,A -85,B 0,C 180,E1 -1673.598,E2 -1673.598} C_VEL
LIN {X 0,Y 580.316,Z 512.193,A -85,B 0,C 180,E1 -1676.146,E2 -1676.146} C_VEL
LIN {X 0,Y 580.283,Z 512.197,A -85,B 0,C 180,E1 -1678.616,E2 -1678.616} C_VEL
LIN {X 0,Y 580.294,Z 512.199,A -85,B 0,C 180,E1 -1681.025,E2 -1681.025} C_VEL
LIN {X 0,Y 580.293,Z 512.201,A -85,B 0,C 180,E1 -1683.667,E2 -1683.667} C_VEL
LIN {X 0,Y 580.3,Z 512.2,A -85,B 0,C 180,E1 -1685.684,E2 -1685.684} C_VEL
LIN {X 0,Y 580.288,Z 512.198,A -85,B 0,C 180,E1 -1688.695,E2 -1688.695} C_VEL
LIN {X 0,Y 580.323,Z 512.196,A -85,B 0,C 180,E1 -1690.915,E2 -1690.915} C_VEL
LIN {X 0,Y 580.284,Z 512.203,A -85,B 0,C 180,E1 -1693.826,E2 -1693.826} C_VEL
LIN {X 0,Y 580.347,Z 512.294,A -85,B 0,C 180,E1 -1694.369,E2 -1694.369} C_VEL
LIN {X 0,Y 580.548,Z 517.414,A -85,B 0,C 180,E1 -1695.273,E2 -1695.273} C_VEL
LIN {X 0,Y 580.405,Z 534.905,A -85,B 0,C 180,E1 -1698.298,E2 -1698.298} C_VEL
LIN {X 0,Y 580.282,Z 547.164,A -85,B 0,C 180,E1 -1700.392,E2 -1700.392} C_VEL
LIN {X 0,Y 580.977,Z 551.646,A -85,B 0,C 180,E1 -1700.47,E2 -1700.47} C_VEL
LIN {X 0,Y 580.801,Z 654.328,A -85,B 0,C 180,E1 -1701.76,E2 -1701.76} C_VEL
LIN {X 0,Y 580.73,Z 667.353,A -85,B 0,C 180,E1 -1702.066,E2 -1702.066} C_VEL
LIN {X 0,Y 580.642,Z 679.351,A -85,B 0,C 180,E1 -1702.48,E2 -1702.48} C_VEL
LIN {X 0,Y 580.569,Z 691.514,A -85,B 0,C 180,E1 -1703.047,E2 -1703.047} C_VEL
LIN {X 0,Y 580.447,Z 703.012,A -85,B 0,C 180,E1 -1703.744,E2 -1703.744} C_VEL
LIN {X 0,Y 580.347,Z 713.356,A -85,B 0,C 180,E1 -1704.528,E2 -1704.528} C_VEL
LIN {X 0,Y 580.317,Z 721.841,A -85,B 0,C 180,E1 -1705.311,E2 -1705.311} C_VEL
LIN {X 0,Y 580.174,Z 729.688,A -85,B 0,C 180,E1 -1706.18,E2 -1706.18} C_VEL
LIN {X 0,Y 580.13,Z 737.37,A -85,B 0,C 180,E1 -1707.223,E2 -1707.223} C_VEL
LIN {X 0,Y 580.134,Z 743.543,A -85,B 0,C 180,E1 -1708.265,E2 -1708.265} C_VEL
LIN {X 0,Y 580.056,Z 748.464,A -85,B 0,C 180,E1 -1709.306,E2 -1709.306} C_VEL
LIN {X 0,Y 580.094,Z 752.273,A -85,B 0,C 180,E1 -1710.347,E2 -1710.347} C_VEL
LIN {X 0,Y 580.047,Z 755.073,A -85,B 0,C 180,E1 -1711.389,E2 -1711.389} C_VEL
LIN {X 0,Y 580.038,Z 757.322,A -85,B 0,C 180,E1 -1712.778,E2 -1712.778} C_VEL
LIN {X 0,Y 580.106,Z 757.864,A -85,B 0,C 180,E1 -1713.473,E2 -1713.473} C_VEL
LIN {X 0,Y 580.087,Z 757.978,A -85,B 0,C 180,E1 -1714.169,E2 -1714.169} C_VEL
LIN {X 0,Y 580.091,Z 757.039,A -85,B 0,C 180,E1 -1715.562,E2 -1715.562} C_VEL
LIN {X 0,Y 580.1,Z 755.362,A -85,B 0,C 180,E1 -1716.562,E2 -1716.562} C_VEL
LIN {X 0,Y 580.081,Z 751.405,A -85,B 0,C 180,E1 -1718.009,E2 -1718.009} C_VEL
LIN {X 0,Y 580.072,Z 747.276,A -85,B 0,C 180,E1 -1719.062,E2 -1719.062} C_VEL
LIN {X 0,Y 580.13,Z 740.933,A -85,B 0,C 180,E1 -1720.293,E2 -1720.293} C_VEL
LIN {X 0,Y 580.194,Z 734.002,A -85,B 0,C 180,E1 -1721.352,E2 -1721.352} C_VEL
LIN {X 0,Y 580.262,Z 726.905,A -85,B 0,C 180,E1 -1722.237,E2 -1722.237} C_VEL
LIN {X 0,Y 580.314,Z 718.304,A -85,B 0,C 180,E1 -1723.125,E2 -1723.125} C_VEL
LIN {X 0,Y 580.431,Z 707.657,A -85,B 0,C 180,E1 -1724.014,E2 -1724.014} C_VEL
LIN {X 0,Y 580.486,Z 697.045,A -85,B 0,C 180,E1 -1724.729,E2 -1724.729} C_VEL
LIN {X 0,Y 580.625,Z 685.269,A -85,B 0,C 180,E1 -1725.353,E2 -1725.353} C_VEL
LIN {X 0,Y 580.695,Z 672.98,A -85,B 0,C 180,E1 -1725.847,E2 -1725.847} C_VEL
LIN {X 0,Y 580.781,Z 660.422,A -85,B 0,C 180,E1 -1726.205,E2 -1726.205} C_VEL
LIN {X 0,Y 580.825,Z 647.769,A -85,B 0,C 180,E1 -1726.429,E2 -1726.429} C_VEL
LIN {X 0,Y 580.881,Z 550.487,A -85,B 0,C 180,E1 -1727.637,E2 -1727.637} C_VEL
LIN {X 0,Y 580.308,Z 547.062,A -85,B 0,C 180,E1 -1727.715,E2 -1727.715} C_VEL
LIN {X 0,Y 580.416,Z 530.458,A -85,B 0,C 180,E1 -1730.557,E2 -1730.557} C_VEL
LIN {X 0,Y 580.577,Z 515.039,A -85,B 0,C 180,E1 -1733.232,E2 -1733.232} C_VEL
LIN {X 0,Y 580.309,Z 512.199,A -85,B 0,C 180,E1 -1733.745,E2 -1733.745} C_VEL
LIN {X 0,Y 580.279,Z 512.207,A -85,B 0,C 180,E1 -1736.623,E2 -1736.623} C_VEL
LIN {X 0,Y 580.302,Z 512.196,A -85,B 0,C 180,E1 -1739.309,E2 -1739.309} C_VEL
LIN {X 0,Y 580.302,Z 512.197,A -85,B 0,C 180,E1 -1742.199,E2 -1742.199} C_VEL
LIN {X 0,Y 580.291,Z 512.206,A -85,B 0,C 180,E1 -1744.695,E2 -1744.695} C_VEL
LIN {X 0,Y 580.3,Z 512.196,A -85,B 0,C 180,E1 -1747.267,E2 -1747.267} C_VEL
LIN {X 0,Y 580.297,Z 512.199,A -85,B 0,C 180,E1 -1750.271,E2 -1750.271} C_VEL
LIN {X 0,Y 580.288,Z 512.206,A -85,B 0,C 180,E1 -1752.704,E2 -1752.704} C_VEL
LIN {X 0,Y 580.27,Z 512.198,A -85,B 0,C 180,E1 -1755.608,E2 -1755.608} C_VEL
LIN {X 0,Y 580.31,Z 512.196,A -85,B 0,C 180,E1 -1758.233,E2 -1758.233} C_VEL
LIN {X 0,Y 580.285,Z 512.202,A -85,B 0,C 180,E1 -1760.965,E2 -1760.965} C_VEL
LIN {X 0,Y 580.291,Z 512.195,A -85,B 0,C 180,E1 -1763.598,E2 -1763.598} C_VEL
LIN {X 0,Y 580.316,Z 512.195,A -85,B 0,C 180,E1 -1766.145,E2 -1766.145} C_VEL
LIN {X 0,Y 580.285,Z 512.206,A -85,B 0,C 180,E1 -1768.615,E2 -1768.615} C_VEL
LIN {X 0,Y 580.29,Z 512.2,A -85,B 0,C 180,E1 -1771.023,E2 -1771.023} C_VEL
LIN {X 0,Y 580.321,Z 512.191,A -85,B 0,C 180,E1 -1773.657,E2 -1773.657} C_VEL
LIN {X 0,Y 580.273,Z 512.205,A -85,B 0,C 180,E1 -1776.442,E2 -1776.442} C_VEL
LIN {X 0,Y 580.275,Z 512.198,A -85,B 0,C 180,E1 -1779.437,E2 -1779.437} C_VEL
LIN {X 0,Y 580.275,Z 512.197,A -85,B 0,C 180,E1 -1781.645,E2 -1781.645} C_VEL
LIN {X 0,Y 580.274,Z 512.198,A -85,B 0,C 180,E1 -1783.825,E2 -1783.825} C_VEL
LIN {X 0,Y 580.316,Z 512.193,A -85,B 0,C 180,E1 -1785.983,E2 -1785.983} C_VEL
LIN {X 0,Y 580.321,Z 512.199,A -85,B 0,C 180,E1 -1788.827,E2 -1788.827} C_VEL
LIN {X 0,Y 580.327,Z 512.19,A -85,B 0,C 180,E1 -1791.644,E2 -1791.644} C_VEL
LIN {X 0,Y 580.318,Z 512.199,A -85,B 0,C 180,E1 -1794.44,E2 -1794.44} C_VEL
LIN {X 0,Y 580.34,Z 512.19,A -85,B 0,C 180,E1 -1797.223,E2 -1797.223} C_VEL
LIN {X 0,Y 580.342,Z 512.19,A -85,B 0,C 180,E1 -1800,E2 -1800} C_VEL
LIN {X 0,Y 580.341,Z 512.196,A -85,B 0,C 180,E1 -1802.776,E2 -1802.776} C_VEL
LIN {X 0,Y 580.317,Z 512.192,A -85,B 0,C 180,E1 -1805.56,E2 -1805.56} C_VEL
LIN {X 0,Y 580.327,Z 512.197,A -85,B 0,C 180,E1 -1808.356,E2 -1808.356} C_VEL
LIN {X 0,Y 580.323,Z 512.193,A -85,B 0,C 180,E1 -1811.208,E2 -1811.208} C_VEL
LIN {X 0,Y 580.304,Z 512.199,A -85,B 0,C 180,E1 -1814.339,E2 -1814.339} C_VEL
LIN {X 0,Y 580.303,Z 512.198,A -85,B 0,C 180,E1 -1816.915,E2 -1816.915} C_VEL
LIN {X 0,Y 580.298,Z 512.195,A -85,B 0,C 180,E1 -1819.823,E2 -1819.823} C_VEL
LIN {X 0,Y 580.266,Z 512.201,A -85,B 0,C 180,E1 -1822.053,E2 -1822.053} C_VEL
LIN {X 0,Y 580.301,Z 512.197,A -85,B 0,C 180,E1 -1825.08,E2 -1825.08} C_VEL
LIN {X 0,Y 580.312,Z 512.193,A -85,B 0,C 180,E1 -1827.864,E2 -1827.864} C_VEL
LIN {X 0,Y 580.291,Z 512.204,A -85,B 0,C 180,E1 -1830.698,E2 -1830.698} C_VEL
LIN {X 0,Y 580.298,Z 512.195,A -85,B 0,C 180,E1 -1833.317,E2 -1833.317} C_VEL
LIN {X 0,Y 580.321,Z 512.192,A -85,B 0,C 180,E1 -1835.768,E2 -1835.768} C_VEL
LIN {X 0,Y 580.282,Z 512.2,A -85,B 0,C 180,E1 -1838.147,E2 -1838.147} C_VEL
LIN {X 0,Y 580.295,Z 512.201,A -85,B 0,C 180,E1 -1840.844,E2 -1840.844} C_VEL
LIN {X 0,Y 580.273,Z 512.198,A -85,B 0,C 180,E1 -1843.659,E2 -1843.659} C_VEL
LIN {X 0,Y 580.282,Z 512.206,A -85,B 0,C 180,E1 -1846.609,E2 -1846.609} C_VEL
LIN {X 0,Y 580.298,Z 512.196,A -85,B 0,C 180,E1 -1849.158,E2 -1849.158} C_VEL
LIN {X 0,Y 580.289,Z 512.198,A -85,B 0,C 180,E1 -1851.927,E2 -1851.927} C_VEL
LIN {X 0,Y 580.277,Z 512.207,A -85,B 0,C 180,E1 -1854.455,E2 -1854.455} C_VEL
LIN {X 0,Y 580.291,Z 512.199,A -85,B 0,C 180,E1 -1856.976,E2 -1856.976} C_VEL
LIN {X 0,Y 580.302,Z 512.195,A -85,B 0,C 180,E1 -1859.426,E2 -1859.426} C_VEL
LIN {X 0,Y 580.299,Z 512.199,A -85,B 0,C 180,E1 -1862.142,E2 -1862.142} C_VEL
LIN {X 0,Y 580.322,Z 512.194,A -85,B 0,C 180,E1 -1865.27,E2 -1865.27} C_VEL
LIN {X 0,Y 580.317,Z 512.365,A -85,B 0,C 180,E1 -1867.106,E2 -1867.106} C_VEL
LIN {X 0,Y 580.919,Z 516.765,A -85,B 0,C 180,E1 -1867.787,E2 -1867.787} C_VEL
LIN {X 0,Y 580.7,Z 536.858,A -85,B 0,C 180,E1 -1870.736,E2 -1870.736} C_VEL
LIN {X 0,Y 580.518,Z 555.803,A -85,B 0,C 180,E1 -1873.471,E2 -1873.471} C_VEL
LIN {X 0,Y 580.384,Z 575.795,A -85,B 0,C 180,E1 -1876.32,E2 -1876.32} C_VEL
LIN {X 0,Y 580.988,Z 581.535,A -85,B 0,C 180,E1 -1876.423,E2 -1876.423} C_VEL
LIN {X 0,Y 580.8,Z 683.962,A -85,B 0,C 180,E1 -1877.708,E2 -1877.708} C_VEL
LIN {X 0,Y 580.738,Z 697.229,A -85,B 0,C 180,E1 -1878.017,E2 -1878.017} C_VEL
LIN {X 0,Y 580.636,Z 710.5,A -85,B 0,C 180,E1 -1878.48,E2 -1878.48} C_VEL
LIN {X 0,Y 580.564,Z 721.635,A -85,B 0,C 180,E1 -1879.009,E2 -1879.009} C_VEL
LIN {X 0,Y 580.426,Z 733.206,A -85,B 0,C 180,E1 -1879.712,E2 -1879.712} C_VEL
LIN {X 0,Y 580.341,Z 743.601,A -85,B 0,C 180,E1 -1880.503,E2 -1880.503} C_VEL
LIN {X 0,Y 580.271,Z 752.114,A -85,B 0,C 180,E1 -1881.292,E2 -1881.292} C_VEL
LIN {X 0,Y 580.221,Z 759.962,A -85,B 0,C 180,E1 -1882.168,E2 -1882.168} C_VEL
LIN {X 0,Y 580.153,Z 767.651,A -85,B 0,C 180,E1 -1883.222,E2 -1883.222} C_VEL
LIN {X 0,Y 580.139,Z 774.681,A -85,B 0,C 180,E1 -1884.439,E2 -1884.439} C_VEL
LIN {X 0,Y 580.108,Z 779.372,A -85,B 0,C 180,E1 -1885.484,E2 -1885.484} C_VEL
LIN {X 0,Y 580.123,Z 782.957,A -85,B 0,C 180,E1 -1886.527,E2 -1886.527} C_VEL
LIN {X 0,Y 580.043,Z 784.809,A -85,B 0,C 180,E1 -1887.222,E2 -1887.222} C_VEL
LIN {X 0,Y 580.038,Z 786.2,A -85,B 0,C 180,E1 -1887.917,E2 -1887.917} C_VEL
LIN {X 0,Y 580.04,Z 787.784,A -85,B 0,C 180,E1 -1889.306,E2 -1889.306} C_VEL
LIN {X 0,Y 580.037,Z 788,A -85,B 0,C 180,E1 -1890,E2 -1890} C_VEL
LIN {X 0,Y 580.047,Z 787.186,A -85,B 0,C 180,E1 -1891.389,E2 -1891.389} C_VEL
LIN {X 0,Y 580.038,Z 786.201,A -85,B 0,C 180,E1 -1892.083,E2 -1892.083} C_VEL
LIN {X 0,Y 580.043,Z 784.81,A -85,B 0,C 180,E1 -1892.778,E2 -1892.778} C_VEL
LIN {X 0,Y 580.109,Z 781.896,A -85,B 0,C 180,E1 -1893.82,E2 -1893.82} C_VEL
LIN {X 0,Y 580.054,Z 777.95,A -85,B 0,C 180,E1 -1894.865,E2 -1894.865} C_VEL
LIN {X 0,Y 580.139,Z 771.878,A -85,B 0,C 180,E1 -1896.085,E2 -1896.085} C_VEL
LIN {X 0,Y 580.184,Z 765.238,A -85,B 0,C 180,E1 -1897.132,E2 -1897.132} C_VEL
LIN {X 0,Y 580.25,Z 756.992,A -85,B 0,C 180,E1 -1898.182,E2 -1898.182} C_VEL
LIN {X 0,Y 580.308,Z 748.54,A -85,B 0,C 180,E1 -1899.058,E2 -1899.058} C_VEL
LIN {X 0,Y 580.415,Z 738.099,A -85,B 0,C 180,E1 -1899.936,E2 -1899.936} C_VEL
LIN {X 0,Y 580.522,Z 727.761,A -85,B 0,C 180,E1 -1900.639,E2 -1900.639} C_VEL
LIN {X 0,Y 580.597,Z 716.237,A -85,B 0,C 180,E1 -1901.264,E2 -1901.264} C_VEL
LIN {X 0,Y 580.662,Z 703.48,A -85,B 0,C 180,E1 -1901.785,E2 -1901.785} C_VEL
LIN {X 0,Y 580.74,Z 690.447,A -85,B 0,C 180,E1 -1902.16,E2 -1902.16} C_VEL
LIN {X 0,Y 580.841,Z 678.106,A -85,B 0,C 180,E1 -1902.38,E2 -1902.38} C_VEL
LIN {X 0,Y 580.876,Z 578.976,A -85,B 0,C 180,E1 -1903.611,E2 -1903.611} C_VEL
LIN {X 0,Y 580.382,Z 575.795,A -85,B 0,C 180,E1 -1903.68,E2 -1903.68} C_VEL
LIN {X 0,Y 580.522,Z 555.803,A -85,B 0,C 180,E1 -1906.529,E2 -1906.529} C_VEL
LIN {X 0,Y 580.701,Z 536.857,A -85,B 0,C 180,E1 -1909.264,E2 -1909.264} C_VEL
LIN {X 0,Y 580.919,Z 516.765,A -85,B 0,C 180,E1 -1912.213,E2 -1912.213} C_VEL
LIN {X 0,Y 580.285,Z 512.204,A -85,B 0,C 180,E1 -1912.926,E2 -1912.926} C_VEL
LIN {X 0,Y 580.306,Z 512.199,A -85,B 0,C 180,E1 -1915.079,E2 -1915.079} C_VEL
LIN {X 0,Y 580.3,Z 512.196,A -85,B 0,C 180,E1 -1918.185,E2 -1918.185} C_VEL
LIN {X 0,Y 580.292,Z 512.196,A -85,B 0,C 180,E1 -1920.695,E2 -1920.695} C_VEL
LIN {X 0,Y 580.304,Z 512.201,A -85,B 0,C 180,E1 -1923.316,E2 -1923.316} C_VEL
LIN {X 0,Y 580.258,Z 512.205,A -85,B 0,C 180,E1 -1925.758,E2 -1925.758} C_VEL
LIN {X 0,Y 580.287,Z 512.197,A -85,B 0,C 180,E1 -1928.145,E2 -1928.145} C_VEL
LIN {X 0,Y 580.298,Z 512.196,A -85,B 0,C 180,E1 -1930.842,E2 -1930.842} C_VEL
LIN {X 0,Y 580.284,Z 512.203,A -85,B 0,C 180,E1 -1933.656,E2 -1933.656} C_VEL
LIN {X 0,Y 580.271,Z 512.198,A -85,B 0,C 180,E1 -1936.609,E2 -1936.609} C_VEL
LIN {X 0,Y 580.295,Z 512.2,A -85,B 0,C 180,E1 -1939.156,E2 -1939.156} C_VEL
LIN {X 0,Y 580.284,Z 512.199,A -85,B 0,C 180,E1 -1941.926,E2 -1941.926} C_VEL
LIN {X 0,Y 580.302,Z 512.194,A -85,B 0,C 180,E1 -1944.456,E2 -1944.456} C_VEL
LIN {X 0,Y 580.285,Z 512.199,A -85,B 0,C 180,E1 -1946.975,E2 -1946.975} C_VEL
LIN {X 0,Y 580.302,Z 512.204,A -85,B 0,C 180,E1 -1949.425,E2 -1949.425} C_VEL
LIN {X 0,Y 580.312,Z 512.194,A -85,B 0,C 180,E1 -1952.136,E2 -1952.136} C_VEL
LIN {X 0,Y 580.301,Z 512.196,A -85,B 0,C 180,E1 -1954.92,E2 -1954.92} C_VEL
LIN {X 0,Y 580.266,Z 512.201,A -85,B 0,C 180,E1 -1957.947,E2 -1957.947} C_VEL
LIN {X 0,Y 580.308,Z 512.195,A -85,B 0,C 180,E1 -1960.914,E2 -1960.914} C_VEL
LIN {X 0,Y 580.273,Z 512.202,A -85,B 0,C 180,E1 -1963.825,E2 -1963.825} C_VEL
LIN {X 0,Y 580.315,Z 512.195,A -85,B 0,C 180,E1 -1965.983,E2 -1965.983} C_VEL
LIN {X 0,Y 580.321,Z 512.193,A -85,B 0,C 180,E1 -1968.827,E2 -1968.827} C_VEL
LIN {X 0,Y 580.327,Z 512.198,A -85,B 0,C 180,E1 -1971.644,E2 -1971.644} C_VEL
LIN {X 0,Y 580.317,Z 512.192,A -85,B 0,C 180,E1 -1974.44,E2 -1974.44} C_VEL
LIN {X 0,Y 580.341,Z 512.196,A -85,B 0,C 180,E1 -1977.224,E2 -1977.224} C_VEL
LIN {X 0,Y 580.342,Z 512.191,A -85,B 0,C 180,E1 -1980,E2 -1980} C_VEL
LIN {X 0,Y 580.34,Z 512.19,A -85,B 0,C 180,E1 -1982.777,E2 -1982.777} C_VEL
LIN {X 0,Y 580.317,Z 512.2,A -85,B 0,C 180,E1 -1985.56,E2 -1985.56} C_VEL
LIN {X 0,Y 580.327,Z 512.191,A -85,B 0,C 180,E1 -1988.356,E2 -1988.356} C_VEL
LIN {X 0,Y 580.323,Z 512.198,A -85,B 0,C 180,E1 -1991.209,E2 -1991.209} C_VEL
LIN {X 0,Y 580.305,Z 512.194,A -85,B 0,C 180,E1 -1994.339,E2 -1994.339} C_VEL
LIN {X 0,Y 580.304,Z 512.196,A -85,B 0,C 180,E1 -1996.915,E2 -1996.915} C_VEL
LIN {X 0,Y 580.299,Z 512.198,A -85,B 0,C 180,E1 -1999.823,E2 -1999.823} C_VEL
LIN {X 0,Y 580.28,Z 512.205,A -85,B 0,C 180,E1 -2001.344,E2 -2001.344} C_VEL
LIN {X 0,Y 579.582,Z 512.287,A -85,B 0,C 180,E1 -2001.923,E2 -2001.923} C_VEL
LIN {X 0,Y 576.704,Z 512.644,A -85,B 0,C 180,E1 -2002.863,E2 -2002.863} C_VEL
LIN {X 0,Y 574.309,Z 512.947,A -85,B 0,C 180,E1 -2003.619,E2 -2003.619} C_VEL
LIN {X 0,Y 573.31,Z 513.066,A -85,B 0,C 180,E1 -2004.203,E2 -2004.203} C_VEL
LIN {X 0,Y 573.243,Z 513.073,A -85,B 0,C 180,E1 -2004.401,E2 -2004.401} C_VEL
LIN {X 0,Y 573.26,Z 513.074,A -85,B 0,C 180,E1 -2006.976,E2 -2006.976} C_VEL
LIN {X 0,Y 573.248,Z 513.082,A -85,B 0,C 180,E1 -2009.491,E2 -2009.491} C_VEL
LIN {X 0,Y 573.25,Z 513.073,A -85,B 0,C 180,E1 -2012.23,E2 -2012.23} C_VEL
LIN {X 0,Y 573.248,Z 513.074,A -85,B 0,C 180,E1 -2014.775,E2 -2014.775} C_VEL
LIN {X 0,Y 573.248,Z 513.079,A -85,B 0,C 180,E1 -2017.167,E2 -2017.167} C_VEL
LIN {X 0,Y 573.243,Z 513.08,A -85,B 0,C 180,E1 -2019.608,E2 -2019.608} C_VEL
LIN {X 0,Y 573.235,Z 513.075,A -85,B 0,C 180,E1 -2022.642,E2 -2022.642} C_VEL
LIN {X 0,Y 573.236,Z 513.08,A -85,B 0,C 180,E1 -2025.668,E2 -2025.668} C_VEL
LIN {X 0,Y 573.244,Z 513.073,A -85,B 0,C 180,E1 -2028.545,E2 -2028.545} C_VEL
LIN {X 0,Y 573.247,Z 513.081,A -85,B 0,C 180,E1 -2031.3,E2 -2031.3} C_VEL
LIN {X 0,Y 573.241,Z 513.075,A -85,B 0,C 180,E1 -2034.015,E2 -2034.015} C_VEL
LIN {X 0,Y 573.269,Z 513.07,A -85,B 0,C 180,E1 -2036.519,E2 -2036.519} C_VEL
LIN {X 0,Y 573.235,Z 513.08,A -85,B 0,C 180,E1 -2039.118,E2 -2039.118} C_VEL
LIN {X 0,Y 573.253,Z 513.074,A -85,B 0,C 180,E1 -2041.972,E2 -2041.972} C_VEL
LIN {X 0,Y 573.255,Z 513.072,A -85,B 0,C 180,E1 -2044.591,E2 -2044.591} C_VEL
LIN {X 0,Y 573.237,Z 513.081,A -85,B 0,C 180,E1 -2047.663,E2 -2047.663} C_VEL
LIN {X 0,Y 573.282,Z 513.071,A -85,B 0,C 180,E1 -2050.729,E2 -2050.729} C_VEL
LIN {X 0,Y 573.256,Z 513.081,A -85,B 0,C 180,E1 -2053.622,E2 -2053.622} C_VEL
LIN {X 0,Y 573.282,Z 513.115,A -85,B 0,C 180,E1 -2054.263,E2 -2054.263} C_VEL
LIN {X 0,Y 573.564,Z 517.718,A -85,B 0,C 180,E1 -2055.089,E2 -2055.089} C_VEL
LIN {X 0,Y 573.382,Z 534.176,A -85,B 0,C 180,E1 -2057.973,E2 -2057.973} C_VEL
LIN {X 0,Y 573.265,Z 547.326,A -85,B 0,C 180,E1 -2060.229,E2 -2060.229} C_VEL
LIN {X 0,Y 574.071,Z 552.144,A -85,B 0,C 180,E1 -2060.309,E2 -2060.309} C_VEL
LIN {X 0,Y 573.875,Z 654.64,A -85,B 0,C 180,E1 -2061.616,E2 -2061.616} C_VEL
LIN {X 0,Y 573.768,Z 667.567,A -85,B 0,C 180,E1 -2061.925,E2 -2061.925} C_VEL
LIN {X 0,Y 573.694,Z 679.505,A -85,B 0,C 180,E1 -2062.344,E2 -2062.344} C_VEL
LIN {X 0,Y 573.619,Z 690.805,A -85,B 0,C 180,E1 -2062.874,E2 -2062.874} C_VEL
LIN {X 0,Y 573.457,Z 702.423,A -85,B 0,C 180,E1 -2063.577,E2 -2063.577} C_VEL
LIN {X 0,Y 573.344,Z 712.906,A -85,B 0,C 180,E1 -2064.372,E2 -2064.372} C_VEL
LIN {X 0,Y 573.285,Z 722.344,A -85,B 0,C 180,E1 -2065.253,E2 -2065.253} C_VEL
LIN {X 0,Y 573.173,Z 731.454,A -85,B 0,C 180,E1 -2066.309,E2 -2066.309} C_VEL
LIN {X 0,Y 573.069,Z 738.8,A -85,B 0,C 180,E1 -2067.364,E2 -2067.364} C_VEL
LIN {X 0,Y 572.985,Z 745.577,A -85,B 0,C 180,E1 -2068.594,E2 -2068.594} C_VEL
LIN {X 0,Y 573.03,Z 750.057,A -85,B 0,C 180,E1 -2069.649,E2 -2069.649} C_VEL
LIN {X 0,Y 572.945,Z 753.472,A -85,B 0,C 180,E1 -2070.703,E2 -2070.703} C_VEL
LIN {X 0,Y 572.947,Z 755.176,A -85,B 0,C 180,E1 -2071.406,E2 -2071.406} C_VEL
LIN {X 0,Y 572.954,Z 757.378,A -85,B 0,C 180,E1 -2072.812,E2 -2072.812} C_VEL
LIN {X 0,Y 573.006,Z 757.886,A -85,B 0,C 180,E1 -2073.516,E2 -2073.516} C_VEL
LIN {X 0,Y 573.007,Z 757.967,A -85,B 0,C 180,E1 -2074.22,E2 -2074.22} C_VEL
LIN {X 0,Y 572.993,Z 756.981,A -85,B 0,C 180,E1 -2075.631,E2 -2075.631} C_VEL
LIN {X 0,Y 573.011,Z 755.451,A -85,B 0,C 180,E1 -2076.549,E2 -2076.549} C_VEL
LIN {X 0,Y 572.994,Z 752.377,A -85,B 0,C 180,E1 -2077.754,E2 -2077.754} C_VEL
LIN {X 0,Y 573.006,Z 748.561,A -85,B 0,C 180,E1 -2078.819,E2 -2078.819} C_VEL
LIN {X 0,Y 573.043,Z 743.598,A -85,B 0,C 180,E1 -2079.886,E2 -2079.886} C_VEL
LIN {X 0,Y 573.128,Z 737.77,A -85,B 0,C 180,E1 -2080.888,E2 -2080.888} C_VEL
LIN {X 0,Y 573.164,Z 730.911,A -85,B 0,C 180,E1 -2081.852,E2 -2081.852} C_VEL
LIN {X 0,Y 573.24,Z 723.182,A -85,B 0,C 180,E1 -2082.749,E2 -2082.749} C_VEL
LIN {X 0,Y 573.321,Z 713.73,A -85,B 0,C 180,E1 -2083.649,E2 -2083.649} C_VEL
LIN {X 0,Y 573.427,Z 702.933,A -85,B 0,C 180,E1 -2084.479,E2 -2084.479} C_VEL
LIN {X 0,Y 573.56,Z 691.433,A -85,B 0,C 180,E1 -2085.183,E2 -2085.183} C_VEL
LIN {X 0,Y 573.723,Z 678.872,A -85,B 0,C 180,E1 -2085.771,E2 -2085.771} C_VEL
LIN {X 0,Y 573.792,Z 665.534,A -85,B 0,C 180,E1 -2086.225,E2 -2086.225} C_VEL
LIN {X 0,Y 573.863,Z 653.455,A -85,B 0,C 180,E1 -2086.497,E2 -2086.497} C_VEL
LIN {X 0,Y 573.981,Z 551.361,A -85,B 0,C 180,E1 -2087.793,E2 -2087.793} C_VEL
LIN {X 0,Y 573.262,Z 547.152,A -85,B 0,C 180,E1 -2087.871,E2 -2087.871} C_VEL
LIN {X 0,Y 573.407,Z 531.217,A -85,B 0,C 180,E1 -2090.632,E2 -2090.632} C_VEL
LIN {X 0,Y 573.591,Z 516.437,A -85,B 0,C 180,E1 -2093.227,E2 -2093.227} C_VEL
LIN {X 0,Y 573.267,Z 513.077,A -85,B 0,C 180,E1 -2093.863,E2 -2093.863} C_VEL
LIN {X 0,Y 573.239,Z 513.083,A -85,B 0,C 180,E1 -2096.492,E2 -2096.492} C_VEL
LIN {X 0,Y 573.24,Z 513.082,A -85,B 0,C 180,E1 -2098.564,E2 -2098.564} C_VEL
LIN {X 0,Y 573.232,Z 513.081,A -85,B 0,C 180,E1 -2100.992,E2 -2100.992} C_VEL
LIN {X 0,Y 573.262,Z 513.072,A -85,B 0,C 180,E1 -2103.523,E2 -2103.523} C_VEL
LIN {X 0,Y 573.244,Z 513.075,A -85,B 0,C 180,E1 -2106.048,E2 -2106.048} C_VEL
LIN {X 0,Y 573.247,Z 513.083,A -85,B 0,C 180,E1 -2108.7,E2 -2108.7} C_VEL
LIN {X 0,Y 573.251,Z 513.073,A -85,B 0,C 180,E1 -2111.595,E2 -2111.595} C_VEL
LIN {X 0,Y 573.236,Z 513.079,A -85,B 0,C 180,E1 -2114.332,E2 -2114.332} C_VEL
LIN {X 0,Y 573.239,Z 513.075,A -85,B 0,C 180,E1 -2117.357,E2 -2117.357} C_VEL
LIN {X 0,Y 573.243,Z 513.078,A -85,B 0,C 180,E1 -2120.392,E2 -2120.392} C_VEL
LIN {X 0,Y 573.251,Z 513.076,A -85,B 0,C 180,E1 -2123.077,E2 -2123.077} C_VEL
LIN {X 0,Y 573.27,Z 513.07,A -85,B 0,C 180,E1 -2125.671,E2 -2125.671} C_VEL
LIN {X 0,Y 573.244,Z 513.076,A -85,B 0,C 180,E1 -2128.184,E2 -2128.184} C_VEL
LIN {X 0,Y 573.264,Z 513.08,A -85,B 0,C 180,E1 -2130.634,E2 -2130.634} C_VEL
LIN {X 0,Y 573.263,Z 513.07,A -85,B 0,C 180,E1 -2133.5,E2 -2133.5} C_VEL
LIN {X 0,Y 573.225,Z 513.078,A -85,B 0,C 180,E1 -2136.134,E2 -2136.134} C_VEL
LIN {X 0,Y 573.253,Z 513.075,A -85,B 0,C 180,E1 -2139.174,E2 -2139.174} C_VEL
LIN {X 0,Y 573.231,Z 513.075,A -85,B 0,C 180,E1 -2141.411,E2 -2141.411} C_VEL
LIN {X 0,Y 573.25,Z 513.072,A -85,B 0,C 180,E1 -2143.622,E2 -2143.622} C_VEL
LIN {X 0,Y 573.229,Z 513.084,A -85,B 0,C 180,E1 -2146.529,E2 -2146.529} C_VEL
LIN {X 0,Y 573.273,Z 513.078,A -85,B 0,C 180,E1 -2148.734,E2 -2148.734} C_VEL
LIN {X 0,Y 573.298,Z 513.066,A -85,B 0,C 180,E1 -2151.541,E2 -2151.541} C_VEL
LIN {X 0,Y 573.284,Z 513.074,A -85,B 0,C 180,E1 -2154.372,E2 -2154.372} C_VEL
LIN {X 0,Y 573.305,Z 513.066,A -85,B 0,C 180,E1 -2157.189,E2 -2157.189} C_VEL
LIN {X 0,Y 573.311,Z 513.066,A -85,B 0,C 180,E1 -2160,E2 -2160} C_VEL
LIN {X 0,Y 573.306,Z 513.071,A -85,B 0,C 180,E1 -2162.811,E2 -2162.811} C_VEL
LIN {X 0,Y 573.284,Z 513.068,A -85,B 0,C 180,E1 -2165.628,E2 -2165.628} C_VEL
LIN {X 0,Y 573.299,Z 513.074,A -85,B 0,C 180,E1 -2168.459,E2 -2168.459} C_VEL
LIN {X 0,Y 573.289,Z 513.069,A -85,B 0,C 180,E1 -2171.312,E2 -2171.312} C_VEL
LIN {X 0,Y 573.27,Z 513.076,A -85,B 0,C 180,E1 -2174.425,E2 -2174.425} C_VEL
LIN {X 0,Y 573.25,Z 513.075,A -85,B 0,C 180,E1 -2177.112,E2 -2177.112} C_VEL
LIN {X 0,Y 573.248,Z 513.075,A -85,B 0,C 180,E1 -2180.077,E2 -2180.077} C_VEL
LIN {X 0,Y 573.229,Z 513.081,A -85,B 0,C 180,E1 -2182.338,E2 -2182.338} C_VEL
LIN {X 0,Y 573.249,Z 513.073,A -85,B 0,C 180,E1 -2185.41,E2 -2185.41} C_VEL
LIN {X 0,Y 573.256,Z 513.073,A -85,B 0,C 180,E1 -2188.032,E2 -2188.032} C_VEL
LIN {X 0,Y 573.236,Z 513.079,A -85,B 0,C 180,E1 -2190.886,E2 -2190.886} C_VEL
LIN {X 0,Y 573.281,Z 513.069,A -85,B 0,C 180,E1 -2193.529,E2 -2193.529} C_VEL
LIN {X 0,Y 573.255,Z 513.075,A -85,B 0,C 180,E1 -2196.049,E2 -2196.049} C_VEL
LIN {X 0,Y 573.243,Z 513.081,A -85,B 0,C 180,E1 -2198.702,E2 -2198.702} C_VEL
LIN {X 0,Y 573.248,Z 513.073,A -85,B 0,C 180,E1 -2201.596,E2 -2201.596} C_VEL
LIN {X 0,Y 573.23,Z 513.082,A -85,B 0,C 180,E1 -2204.334,E2 -2204.334} C_VEL
LIN {X 0,Y 573.24,Z 513.074,A -85,B 0,C 180,E1 -2207.359,E2 -2207.359} C_VEL
LIN {X 0,Y 573.245,Z 513.081,A -85,B 0,C 180,E1 -2210.394,E2 -2210.394} C_VEL
LIN {X 0,Y 573.251,Z 513.075,A -85,B 0,C 180,E1 -2213.079,E2 -2213.079} C_VEL
LIN {X 0,Y 573.266,Z 513.071,A -85,B 0,C 180,E1 -2215.672,E2 -2215.672} C_VEL
LIN {X 0,Y 573.248,Z 513.078,A -85,B 0,C 180,E1 -2218.186,E2 -2218.186} C_VEL
LIN {X 0,Y 573.264,Z 513.08,A -85,B 0,C 180,E1 -2220.635,E2 -2220.635} C_VEL
LIN {X 0,Y 573.251,Z 513.077,A -85,B 0,C 180,E1 -2223.025,E2 -2223.025} C_VEL
LIN {X 0,Y 573.276,Z 513.072,A -85,B 0,C 180,E1 -2225.367,E2 -2225.367} C_VEL
LIN {X 0,Y 573.254,Z 513.218,A -85,B 0,C 180,E1 -2226.937,E2 -2226.937} C_VEL
LIN {X 0,Y 574.016,Z 518.024,A -85,B 0,C 180,E1 -2227.695,E2 -2227.695} C_VEL
LIN {X 0,Y 573.749,Z 538.173,A -85,B 0,C 180,E1 -2230.687,E2 -2230.687} C_VEL
LIN {X 0,Y 573.541,Z 557.107,A -85,B 0,C 180,E1 -2233.454,E2 -2233.454} C_VEL
LIN {X 0,Y 573.433,Z 576.169,A -85,B 0,C 180,E1 -2236.173,E2 -2236.173} C_VEL
LIN {X 0,Y 574.086,Z 581.535,A -85,B 0,C 180,E1 -2236.257,E2 -2236.257} C_VEL
LIN {X 0,Y 573.877,Z 683.962,A -85,B 0,C 180,E1 -2237.558,E2 -2237.558} C_VEL
LIN {X 0,Y 573.794,Z 697.229,A -85,B 0,C 180,E1 -2237.87,E2 -2237.87} C_VEL
LIN {X 0,Y 573.688,Z 710.501,A -85,B 0,C 180,E1 -2238.339,E2 -2238.339} C_VEL
LIN {X 0,Y 573.576,Z 721.726,A -85,B 0,C 180,E1 -2238.879,E2 -2238.879} C_VEL
LIN {X 0,Y 573.437,Z 733.207,A -85,B 0,C 180,E1 -2239.585,E2 -2239.585} C_VEL
LIN {X 0,Y 573.326,Z 743.602,A -85,B 0,C 180,E1 -2240.386,E2 -2240.386} C_VEL
LIN {X 0,Y 573.241,Z 752.115,A -85,B 0,C 180,E1 -2241.185,E2 -2241.185} C_VEL
LIN {X 0,Y 573.161,Z 759.962,A -85,B 0,C 180,E1 -2242.071,E2 -2242.071} C_VEL
LIN {X 0,Y 573.072,Z 767.955,A -85,B 0,C 180,E1 -2243.186,E2 -2243.186} C_VEL
LIN {X 0,Y 573.07,Z 774.681,A -85,B 0,C 180,E1 -2244.37,E2 -2244.37} C_VEL
LIN {X 0,Y 573.029,Z 779.372,A -85,B 0,C 180,E1 -2245.428,E2 -2245.428} C_VEL
LIN {X 0,Y 573.022,Z 782.957,A -85,B 0,C 180,E1 -2246.484,E2 -2246.484} C_VEL
LIN {X 0,Y 572.959,Z 784.808,A -85,B 0,C 180,E1 -2247.188,E2 -2247.188} C_VEL
LIN {X 0,Y 572.937,Z 786.199,A -85,B 0,C 180,E1 -2247.891,E2 -2247.891} C_VEL
LIN {X 0,Y 572.941,Z 787.785,A -85,B 0,C 180,E1 -2249.297,E2 -2249.297} C_VEL
LIN {X 0,Y 572.938,Z 788,A -85,B 0,C 180,E1 -2250,E2 -2250} C_VEL
LIN {X 0,Y 572.946,Z 787.186,A -85,B 0,C 180,E1 -2251.406,E2 -2251.406} C_VEL
LIN {X 0,Y 572.937,Z 786.2,A -85,B 0,C 180,E1 -2252.109,E2 -2252.109} C_VEL
LIN {X 0,Y 572.959,Z 784.81,A -85,B 0,C 180,E1 -2252.812,E2 -2252.812} C_VEL
LIN {X 0,Y 573.014,Z 781.896,A -85,B 0,C 180,E1 -2253.868,E2 -2253.868} C_VEL
LIN {X 0,Y 572.963,Z 777.95,A -85,B 0,C 180,E1 -2254.925,E2 -2254.925} C_VEL
LIN {X 0,Y 573.064,Z 771.878,A -85,B 0,C 180,E1 -2256.16,E2 -2256.16} C_VEL
LIN {X 0,Y 573.119,Z 765.239,A -85,B 0,C 180,E1 -2257.221,E2 -2257.221} C_VEL
LIN {X 0,Y 573.201,Z 756.992,A -85,B 0,C 180,E1 -2258.283,E2 -2258.283} C_VEL
LIN {X 0,Y 573.286,Z 748.541,A -85,B 0,C 180,E1 -2259.17,E2 -2259.17} C_VEL
LIN {X 0,Y 573.42,Z 738.1,A -85,B 0,C 180,E1 -2260.058,E2 -2260.058} C_VEL
LIN {X 0,Y 573.546,Z 726.357,A -85,B 0,C 180,E1 -2260.858,E2 -2260.858} C_VEL
LIN {X 0,Y 573.652,Z 715.287,A -85,B 0,C 180,E1 -2261.447,E2 -2261.447} C_VEL
LIN {X 0,Y 573.748,Z 702.182,A -85,B 0,C 180,E1 -2261.974,E2 -2261.974} C_VEL
LIN {X 0,Y 573.836,Z 689.532,A -85,B 0,C 180,E1 -2262.331,E2 -2262.331} C_VEL
LIN {X 0,Y 573.931,Z 676.334,A -85,B 0,C 180,E1 -2262.553,E2 -2262.553} C_VEL
LIN {X 0,Y 573.959,Z 579.746,A -85,B 0,C 180,E1 -2263.769,E2 -2263.769} C_VEL
LIN {X 0,Y 573.379,Z 575.795,A -85,B 0,C 180,E1 -2263.851,E2 -2263.851} C_VEL
LIN {X 0,Y 573.543,Z 555.893,A -85,B 0,C 180,E1 -2266.722,E2 -2266.722} C_VEL
LIN {X 0,Y 573.734,Z 537.582,A -85,B 0,C 180,E1 -2269.4,E2 -2269.4} C_VEL
